    // Приоритет 2: Датчики движения (ТЗ 2.0)
    // Защита от дребезга и удержание сигнала движения с помощью TOF
    L_Motion_Timers[L_i](IN := VI_Motion_Sensors[L_i], PT := T#5m, VI_System_Time_MS := VI_System_Time_MS);
    
    // Сброс ручного переопределения, когда комната становится пустой (задний фронт таймера движения)
    IF L_Prev_Motion_Q[L_i] AND NOT L_Motion_Timers[L_i].Q THEN
        L_Manual_Override[L_i] := FALSE;
    END_IF;
    L_Prev_Motion_Q[L_i] := L_Motion_Timers[L_i].Q;

    IF L_Motion_Timers[L_i].Q THEN
        IF NOT L_Manual_Override[L_i] THEN
            L_Light_States[L_i] := TRUE;
        END_IF;
    ELSE
        // Выключаем свет только если нет ручного переопределения
        IF NOT L_Manual_Override[L_i] THEN
            L_Light_States[L_i] := FALSE;
        END_IF;
    END_IF;

    // Приоритет 3: Симуляция (только в режиме Away)
    IF L_Effective_Scenario = E_SCENARIO_TYPE.SCENARIO_AWAY AND L_Effective_Simulation_Active THEN
        L_Light_States[L_i] := VI_Simulation_Lights[L_i];
    END_IF;

    // Приоритет 4: Ручное управление и правила
    IF VI_Manual_Light_Override[L_i] > 0 THEN
        VO_Lighting_Levels[L_i] := VI_Manual_Light_Override[L_i];
    ELSIF L_Rule_Light_Active THEN
        VO_Lighting_Levels[L_i] := L_Rule_Light_Val;
    ELSE
        VO_Lighting_Levels[L_i] := SEL(L_Light_States[L_i], 0, L_Base_Light);
    END_IF;
    
    // 5. Мокрые зоны
    IF VI_Wet_Zone_Map[L_i] AND L_Wet_Zone_Idx <= GVL_CONSTANTS.C_MAX_WET_ZONES THEN
        VO_Wet_Zone_Light_Active[L_Wet_Zone_Idx] := (VO_Lighting_Levels[L_i] > 10);
        L_Wet_Zone_Idx := L_Wet_Zone_Idx + 1;
    END_IF;
END_FOR;

// 3. Управление шторами
FOR L_i := 1 TO GVL_CONSTANTS.C_MAX_BLINDS DO
    L_Rule_Blinds_Active := FALSE;
    L_Rule_Blinds_Val := 0;
    
    // Проверка правил
    FOR L_j := 1 TO GVL_CONSTANTS.C_MAX_RULES DO
        IF VI_Rule_Actions[L_j].Active AND VI_Rule_Actions[L_j].Target_ID = L_i THEN
            IF VI_Rule_Actions[L_j].Action_Type = E_Rule_Action_Type.ACTION_SET_BLINDS THEN
                L_Rule_Blinds_Active := TRUE;
                L_Rule_Blinds_Val := REAL_TO_BYTE(VI_Rule_Actions[L_j].Value);
            END_IF;
        END_IF;
    END_FOR;

    // Приоритет 1: Ручное управление
    IF VI_Manual_Blinds_Override[L_i] > 0 THEN
        VO_Blinds_Positions[L_i] := VI_Manual_Blinds_Override[L_i];
    // Приоритет 2: Правила
    ELSIF L_Rule_Blinds_Active THEN
        VO_Blinds_Positions[L_i] := L_Rule_Blinds_Val;
    // Приоритет 3: Сценарий
    ELSE
        VO_Blinds_Positions[L_i] := L_Base_Blinds;
    END_IF;
END_FOR;

// >>> BULK_SYNC_ANCHOR: FB_Lighting_Blinds_Manager <<<
          
END_FUNCTION_BLOCK

FUNCTION_BLOCK FB_Trace_Logger
  VAR_INPUT
    VI_Event_Code : INT;
    VI_System_Time : UDINT;
  END_VAR

            GVL_TRACE.G_Trace_Index := GVL_TRACE.G_Trace_Index + 1;
IF GVL_TRACE.G_Trace_Index > GVL_TRACE.G_Trace_Max THEN
    GVL_TRACE.G_Trace_Index := 1;
END_IF;

GVL_TRACE.G_Trace_Time[GVL_TRACE.G_Trace_Index] := VI_System_Time;
GVL_TRACE.G_Trace_Code[GVL_TRACE.G_Trace_Index] := VI_Event_Code;
          
END_FUNCTION_BLOCK

FUNCTION_BLOCK FB_Heating_System_Manager
  VAR_INPUT
    VI_Preheat_Request : BOOL;
    L_Climate_Zone_ID : INT;
    VI_System_Mode : E_System_Operating_Mode;
    VI_System_Time_MS : UDINT;
    VI_Current_TOD : TOD;
    VI_IsActivePLC : BOOL;
    VI_Outdoor_Temp : REAL;
    VI_Config : ST_Heating_Config;
    VI_Tariff : ST_Tariff_Config;
    VI_Current_Hour : UINT;
    VI_Boiler_Stop : BOOL;
    VI_DHW_Heating_Demand : BOOL;
    VI_DHW_Target_Temp : REAL;
    VI_Current_Scenario : E_SCENARIO_TYPE;
    VI_Emergency_Stop : BOOL;
    VI_Gas_Safety_Stop : BOOL;
    VI_Boiler_Error_Status : ARRAY[1..GVL_CONSTANTS.C_MAX_BOILERS] OF BOOL;
    VI_Boiler_OT_Online : ARRAY[1..GVL_CONSTANTS.C_MAX_BOILERS] OF BOOL;
    VI_Boiler_Modulation : ARRAY[1..GVL_CONSTANTS.C_MAX_BOILERS] OF REAL;
  END_VAR
  VAR_OUTPUT
    VO_Manifold_Valves : ARRAY[1..GVL_CONSTANTS.C_MAX_MANIFOLDS] OF REAL;
    VO_Manifold_Pumps : ARRAY[1..GVL_CONSTANTS.C_MAX_MANIFOLDS] OF BOOL;
    VO_Zone_Valves : ARRAY[1..GVL_CONSTANTS.C_MAX_HEATING_CIRCUITS] OF BOOL;
    VO_Boiler_OT_Enable : ARRAY[1..GVL_CONSTANTS.C_MAX_BOILERS] OF BOOL;
    VO_Boiler_OT_Setpoint : ARRAY[1..GVL_CONSTANTS.C_MAX_BOILERS] OF REAL;
    VO_Backup_Circulation_Pump : BOOL;
    VO_Electric_Heater_Enable : BOOL;
    VO_Freeze_Risk_Status : BOOL;
    VO_Status : ARRAY[1..GVL_CONSTANTS.C_MAX_MANIFOLDS] OF ST_Manifold_Status;
    VO_Boiler_Status : ARRAY[1..GVL_CONSTANTS.C_MAX_BOILERS] OF ST_Boiler_Status;
  END_VAR
  VAR_IN_OUT
    VI_Floor_Temps : ARRAY[1..GVL_CONSTANTS.C_MAX_HEATING_CIRCUITS] OF REAL;
    VI_Room_Temps : ARRAY[1..16] OF REAL;
    VI_Manifold_Pressures : ARRAY[1..GVL_CONSTANTS.C_MAX_MANIFOLDS] OF REAL;
    VI_Manifold_Currents : ARRAY[1..GVL_CONSTANTS.C_MAX_MANIFOLDS] OF REAL;
    VI_Manifold_Temps_Supply : ARRAY[1..GVL_CONSTANTS.C_MAX_MANIFOLDS] OF REAL;
    VI_Manifold_Temps_Return : ARRAY[1..GVL_CONSTANTS.C_MAX_MANIFOLDS] OF REAL;
    VI_Boiler_Flame_Status : ARRAY[1..GVL_CONSTANTS.C_MAX_BOILERS] OF BOOL;
    VI_Zone_Configs : ARRAY[1..GVL_CONSTANTS.C_MAX_HEATING_CIRCUITS] OF ST_FloorHeating_Circuit_Config;
    VI_Rule_Actions : ARRAY[1..GVL_CONSTANTS.C_MAX_RULES] OF ST_Rule_Action;
    VI_IO_Modules_Online : ARRAY[1..GVL_CONSTANTS.C_MAX_MODULES] OF BOOL;
    VI_Scenario_Configs : ARRAY[1..GVL_CONSTANTS.C_MAX_SCENARIOS] OF ST_Scenario_Config;
    VI_Manifold_End_Switches : ARRAY[1..GVL_CONSTANTS.C_MAX_MANIFOLDS] OF BOOL;
    VI_Valve_Test_Config : ARRAY[1..GVL_CONSTANTS.C_MAX_MANIFOLDS] OF ST_Valve_Test_Config;
  END_VAR
  VAR
    L_Lead_Boiler : BYTE := 1;
    L_i : INT;
    L_j : INT;
    L_Target_Supply_Temp : REAL;
    L_Demand_Power : REAL;
    L_Any_Zone_Active : ARRAY[1..GVL_CONSTANTS.C_MAX_MANIFOLDS] OF BOOL;
    L_Prev_Scenario : E_SCENARIO_TYPE;
    L_Scenario_Adjust : REAL;
    L_Target_Scenario_Adjust : REAL;
    L_Transition_Temp : FB_Scenario_Transition_Controller;
    fbValveTestManager : FB_Valve_Test_Manager;
    L_IO_Failsafe_Active : BOOL;
    L_Freeze_Mode_Active : BOOL;
    L_Freeze_Target_Supply : REAL;
    L_Min_Supply_Temp : REAL;
    L_Policy_Degraded : BOOL;
    L_Any_Sensor_Error : BOOL;
    L_Any_Subsystem_Degraded : BOOL;
    L_Adaptive_Max_Delta : REAL;
    L_Adaptive_Effective_Delta : REAL;
    L_Adaptive_Correction : REAL;
    fbAdaptiveTarget : FB_Heating_Adaptive_Target;
    fbSafetyGate : FB_Heating_Safety_Gate;
    fbCircuitControl : FB_Heating_Circuit_Control;
    fbManifoldControl : FB_Heating_Manifold_Control;
    fbBoilerControl : FB_Heating_Boiler_Control;
  END_VAR

            // ==============================================================================
// Блок управления системой отопления (Heating System Manager)
// Назначение:
// - Публичный фасад системы отопления.
// - Оркестрация доменных FB отопления.
// - Проекция безопасных состояний на физические выходы.
// - Интеграция с Rule Engine, HMI status и GVL_STATE.
// ==============================================================================



// ========================================
// Policy and fault pre-scan
// ========================================
L_Policy_Degraded := (VI_System_Mode = E_System_Operating_Mode.MODE_DEGRADED);

GVL_STATE.G_Heating_IO_Fault := FALSE;
GVL_STATE.G_Heating_Sensor_Fault := FALSE;
GVL_STATE.G_Heating_Subsystem_Degraded := FALSE;
L_Any_Sensor_Error := FALSE;
L_Any_Subsystem_Degraded := FALSE;

L_IO_Failsafe_Active := FALSE;
FOR L_i := 1 TO GVL_CONSTANTS.C_MAX_MODULES DO
    IF NOT VI_IO_Modules_Online[L_i] THEN
        L_IO_Failsafe_Active := TRUE;
        GVL_STATE.G_Heating_IO_Fault := TRUE;
        GVL_STATE.G_Heating_Subsystem_Degraded := TRUE;
        EXIT;
    END_IF;
END_FOR;

fbSafetyGate(
    VI_System_Mode := VI_System_Mode,
    VI_Emergency_Stop := VI_Emergency_Stop,
    VI_Gas_Safety_Stop := VI_Gas_Safety_Stop,
    VI_IO_Failsafe_Active := L_IO_Failsafe_Active,
    VI_Outdoor_Temp := VI_Outdoor_Temp,
    VI_Freeze_Threshold := VI_Config.Freeze_Threshold,
    VI_Floor_Temps := VI_Floor_Temps,
    VO_Freeze_Mode_Active => L_Freeze_Mode_Active,
    VO_Freeze_Target_Supply => L_Freeze_Target_Supply
);

// ========================================
// Safe-state output projection
// ========================================
VO_Backup_Circulation_Pump := FALSE;
VO_Electric_Heater_Enable := FALSE;
VO_Freeze_Risk_Status := FALSE;

IF fbSafetyGate.VO_Block_Normal_Heating THEN
    FOR L_i := 1 TO GVL_CONSTANTS.C_MAX_HEATING_CIRCUITS DO
        VO_Zone_Valves[L_i] := FALSE;
    END_FOR;

    FOR L_i := 1 TO GVL_CONSTANTS.C_MAX_MANIFOLDS DO
        IF fbSafetyGate.VO_IO_Failsafe_Active AND L_Freeze_Mode_Active THEN
            VO_Manifold_Pumps[L_i] := TRUE;
            VO_Manifold_Valves[L_i] := 35.0;
        ELSE
            VO_Manifold_Pumps[L_i] := FALSE;
            VO_Manifold_Valves[L_i] := 0.0;
        END_IF;
    END_FOR;

    FOR L_i := 1 TO GVL_CONSTANTS.C_MAX_BOILERS DO
        VO_Boiler_OT_Enable[L_i] := FALSE;
        VO_Boiler_OT_Setpoint[L_i] := 0.0;
        VO_Boiler_Status[L_i].Warning := FALSE;
        VO_Boiler_Status[L_i].Error := TRUE;
    END_FOR;

    IF fbSafetyGate.VO_Gas_Safety_Active AND L_Freeze_Mode_Active THEN
        VO_Backup_Circulation_Pump := TRUE;
        L_Min_Supply_Temp := 1000.0;
        FOR L_i := 1 TO GVL_CONSTANTS.C_MAX_MANIFOLDS DO
            IF VI_Manifold_Temps_Supply[L_i] < L_Min_Supply_Temp THEN
                L_Min_Supply_Temp := VI_Manifold_Temps_Supply[L_i];
            END_IF;
        END_FOR;
        IF L_Min_Supply_Temp > 900.0 THEN
            L_Min_Supply_Temp := 0.0;
        END_IF;

        IF L_Min_Supply_Temp < (L_Freeze_Target_Supply - 1.0) THEN
            VO_Electric_Heater_Enable := TRUE;
        ELSIF L_Min_Supply_Temp > (L_Freeze_Target_Supply + 1.0) THEN
            VO_Electric_Heater_Enable := FALSE;
        END_IF;

        // При защёлкнутой газовой аварии оператор должен видеть, что система живёт в деградированном anti-freeze режиме.
        VO_Freeze_Risk_Status := TRUE;
    END_IF;

    IF fbSafetyGate.VO_IO_Failsafe_Active AND L_Freeze_Mode_Active THEN
        IF VI_Boiler_OT_Online[1] AND NOT VI_Boiler_Error_Status[1] THEN
            VO_Boiler_OT_Enable[1] := TRUE;
            VO_Boiler_OT_Setpoint[1] := L_Freeze_Target_Supply;
        END_IF;
    END_IF;

    RETURN;
END_IF;

// --- ADAPTIVE TARGET ---
fbAdaptiveTarget(
    VI_Base_Target_Supply_Temp := L_Target_Supply_Temp,
    VI_Global_Target_Temperature := GVL_STATE.G_Target_Temperature,
    VI_Zone_Configs := VI_Zone_Configs,
    VI_Floor_Temps := VI_Floor_Temps,
    VI_Room_Temps := VI_Room_Temps,
    VO_Target_Supply_Temp => L_Target_Supply_Temp,
    VO_Adaptive_Correction => L_Adaptive_Correction,
    VO_Adaptive_Effective_Delta => L_Adaptive_Effective_Delta,
    VO_Adaptive_Max_Delta => L_Adaptive_Max_Delta
);

// --- CIRCUIT CONTROL ---
fbCircuitControl(
    VI_System_Time_MS := VI_System_Time_MS,
    VI_Current_Hour := VI_Current_Hour,
    VI_IsActivePLC := VI_IsActivePLC,
    VI_Config := VI_Config,
    VI_Tariff := VI_Tariff,
    VI_Scenario_Adjust := L_Scenario_Adjust,
    VI_Zone_Configs := VI_Zone_Configs,
    VI_Floor_Temps := VI_Floor_Temps,
    VI_Room_Temps := VI_Room_Temps,
    VI_Rule_Actions := VI_Rule_Actions,
    VO_Zone_Valves => VO_Zone_Valves,
    VO_Heating_Sensor_Fault => L_Any_Sensor_Error
);

GVL_STATE.G_Heating_Sensor_Fault := L_Any_Sensor_Error;

// --- MANIFOLD DEMAND MAP ---
FOR L_i := 1 TO GVL_CONSTANTS.C_MAX_MANIFOLDS DO
    L_Any_Zone_Active[L_i] := FALSE;
END_FOR;

FOR L_i := 1 TO GVL_CONSTANTS.C_MAX_HEATING_CIRCUITS DO
    IF VO_Zone_Valves[L_i] THEN
        L_j := VI_Zone_Configs[L_i].manifold_id;
        IF L_j >= 1 AND L_j <= GVL_CONSTANTS.C_MAX_MANIFOLDS THEN
            L_Any_Zone_Active[L_j] := TRUE;
        END_IF;
    END_IF;
END_FOR;

// --- MANIFOLD CONTROL ---
fbManifoldControl(
    VI_System_Time_MS := VI_System_Time_MS,
    VI_IsActivePLC := VI_IsActivePLC,
    VI_DHW_Heating_Demand := VI_DHW_Heating_Demand,
    VI_Freeze_Mode_Active := L_Freeze_Mode_Active,
    VI_Target_Supply_Temp := L_Target_Supply_Temp,
    VI_Any_Zone_Active := L_Any_Zone_Active,
    VI_Manifold_Pressures := VI_Manifold_Pressures,
    VI_Manifold_Currents := VI_Manifold_Currents,
    VI_Manifold_Temps_Supply := VI_Manifold_Temps_Supply,
    VI_Manifold_Temps_Return := VI_Manifold_Temps_Return,
    VO_Manifold_Pumps => VO_Manifold_Pumps,
    VO_Manifold_Valves => VO_Manifold_Valves,
    VO_Status => VO_Status
);

// --- VALVE TEST OVERRIDE ---
fbValveTestManager(
    VI_System_Time_MS := VI_System_Time_MS,
    VI_IsActivePLC := VI_IsActivePLC,
    VI_Valve_Currents := VI_Manifold_Currents,
    VI_Valve_End_Switches := VI_Manifold_End_Switches,
    VI_Config := VI_Valve_Test_Config
);

IF fbValveTestManager.VO_Test_Active THEN
    L_i := fbValveTestManager.VO_Current_Valve;
    IF L_i >= 1 AND L_i <= GVL_CONSTANTS.C_MAX_MANIFOLDS THEN
        IF fbValveTestManager.VO_Valve_Cmd[L_i] THEN
            VO_Manifold_Valves[L_i] := 100.0;
        ELSE
            VO_Manifold_Valves[L_i] := 0.0;
        END_IF;
        VO_Manifold_Pumps[L_i] := FALSE; // Отключаем насос при тестировании клапана
    END_IF;
END_IF;

// --- BOILER CONTROL ---
fbBoilerControl(
    VI_System_Time_MS := VI_System_Time_MS,
    VI_IsActivePLC := VI_IsActivePLC,
    VI_DHW_Heating_Demand := VI_DHW_Heating_Demand,
    VI_DHW_Target_Temp := VI_DHW_Target_Temp,
    VI_Target_Supply_Temp := L_Target_Supply_Temp,
    VI_Freeze_Mode_Active := L_Freeze_Mode_Active,
    VI_Policy_Degraded := L_Policy_Degraded,
    VI_Manifold_Pumps := VO_Manifold_Pumps,
    VI_Manifold_Valves := VO_Manifold_Valves,
    VI_Boiler_Flame_Status := VI_Boiler_Flame_Status,
    VI_Boiler_Error_Status := VI_Boiler_Error_Status,
    VI_Boiler_OT_Online := VI_Boiler_OT_Online,
    VI_Boiler_Modulation := VI_Boiler_Modulation,
    VO_Boiler_OT_Enable => VO_Boiler_OT_Enable,
    VO_Boiler_OT_Setpoint => VO_Boiler_OT_Setpoint,
    VO_Boiler_Status => VO_Boiler_Status,
    VO_Any_Subsystem_Degraded => L_Any_Subsystem_Degraded,
    VO_Lead_Boiler => L_Lead_Boiler,
    VO_Demand_Power => L_Demand_Power
);

GVL_STATE.G_Heating_Subsystem_Degraded := L_Any_Subsystem_Degraded;

// >>> BULK_SYNC_ANCHOR: FB_Heating_System_Manager <<<
          
END_FUNCTION_BLOCK

FUNCTION_BLOCK FB_Water_Leakage_Manager
  VAR_INPUT
    VI_System_Time_MS : UDINT;
    VI_IsActivePLC : BOOL;
    VI_Config : ST_Flood_Global_Config;
  END_VAR
  VAR_OUTPUT
    VO_Status_Msg : STRING(200);
    VO_Leak_Detected : BOOL;
    VO_Leak_Warning_Level : BOOL;
  END_VAR
  VAR_IN_OUT
    VI_Sensors : ARRAY[1..GVL_CONSTANTS.C_MAX_FLOOD_SENSORS] OF BOOL;
  END_VAR
  VAR
    L_i : INT;
    L_Sensor_Timers : ARRAY[1..GVL_CONSTANTS.C_MAX_FLOOD_SENSORS] OF FB_System_Timer;
    L_Any_Leak : BOOL;
    L_Any_Warning : BOOL;
  END_VAR

            IF NOT VI_IsActivePLC THEN RETURN; END_IF;

L_Any_Leak := FALSE;
L_Any_Warning := FALSE;

FOR L_i := 1 TO GVL_CONSTANTS.C_MAX_FLOOD_SENSORS DO
    L_Sensor_Timers[L_i](
        IN := VI_Sensors[L_i],
        PT := TO_TIME(VI_Config.min_duration_ms + VI_Config.warning_duration_ms),
        VI_System_Time_MS := VI_System_Time_MS
    );

    IF L_Sensor_Timers[L_i].ET >= TO_TIME(VI_Config.min_duration_ms) THEN
        L_Any_Warning := TRUE;

        IF L_Sensor_Timers[L_i].Q THEN
            L_Any_Leak := TRUE;
        END_IF;
    END_IF;
END_FOR;

// Health signals
VO_Leak_Detected := L_Any_Leak;
VO_Leak_Warning_Level := L_Any_Warning;

// Status
IF L_Any_Leak THEN
    VO_Status_Msg := 'АВАРИЯ: ПРОТЕЧКА ВОДЫ.';
ELSIF L_Any_Warning THEN
    VO_Status_Msg := 'ПРЕДУПРЕЖДЕНИЕ: ОБНАРУЖЕНА ВОДА.';
ELSE
    VO_Status_Msg := 'Система контроля протечек в норме';
END_IF;
// >>> BULK_SYNC_ANCHOR: FB_Water_Leakage_Manager <<<
          
END_FUNCTION_BLOCK

FUNCTION_BLOCK FB_Heating_Policy_Observer
  VAR_INPUT
    VI_Zone_Occupied : ARRAY[1..GVL_CONSTANTS.C_MAX_ZONES] OF BOOL;
    VI_Zone_Last_Motion_TS : ARRAY[1..GVL_CONSTANTS.C_MAX_ZONES] OF UDINT;
    VI_System_Time_MS : UDINT;
    VI_Zone_Permanent_Use : ARRAY[1..GVL_CONSTANTS.C_MAX_ZONES] OF BOOL;
    VI_Zone_Guest_Preheat : ARRAY[1..GVL_CONSTANTS.C_MAX_ZONES] OF BOOL;
    VI_Behavior_Mode : E_Behavior_Mode;
  END_VAR
  VAR_OUTPUT
    VO_Zone_Empty_Duration_MS : ARRAY[1..GVL_CONSTANTS.C_MAX_ZONES] OF UDINT;
    VO_Zone_Policy_Class : ARRAY[1..GVL_CONSTANTS.C_MAX_ZONES] OF INT;
    VO_Zone_Target_Adjustment : ARRAY[1..GVL_CONSTANTS.C_MAX_ZONES] OF REAL;
    VO_Zone_Priority_Bias : ARRAY[1..GVL_CONSTANTS.C_MAX_ZONES] OF REAL;
  END_VAR
  VAR
    L_i : INT;
    L_Long_Threshold : UDINT := 86400000;
    L_Away_Mode : BOOL;
  END_VAR

            L_Away_Mode := (VI_Behavior_Mode = BEHAVIOR_AWAY);

FOR L_i := 1 TO GVL_CONSTANTS.C_MAX_ZONES DO

    // compute empty duration
    IF VI_Zone_Occupied[L_i] THEN
        VO_Zone_Empty_Duration_MS[L_i] := 0;
    ELSE
        VO_Zone_Empty_Duration_MS[L_i] := VI_System_Time_MS - VI_Zone_Last_Motion_TS[L_i];
    END_IF;

    // policy classification
    // Guest/preheat has priority even in AWAY mode.
    IF VI_Zone_Guest_Preheat[L_i] THEN
        VO_Zone_Policy_Class[L_i] := 3; // guest

    ELSIF VI_Zone_Occupied[L_i] THEN
        VO_Zone_Policy_Class[L_i] := 0; // comfort

    ELSIF VI_Zone_Permanent_Use[L_i] AND (NOT L_Away_Mode) THEN
        VO_Zone_Policy_Class[L_i] := 4; // permanent mild eco

    ELSIF VO_Zone_Empty_Duration_MS[L_i] >= L_Long_Threshold THEN
        VO_Zone_Policy_Class[L_i] := 2; // deep eco

    ELSE
        VO_Zone_Policy_Class[L_i] := 1; // mild eco
    END_IF;

    // observe-only target adjustment (no effect yet)
    CASE VO_Zone_Policy_Class[L_i] OF
        0: // comfort
            VO_Zone_Target_Adjustment[L_i] := 0.0;
            VO_Zone_Priority_Bias[L_i] := 1.0;

        1: // mild eco
            VO_Zone_Target_Adjustment[L_i] := -1.0;
            VO_Zone_Priority_Bias[L_i] := 0.8;

        2: // deep eco
            VO_Zone_Target_Adjustment[L_i] := -3.0;
            VO_Zone_Priority_Bias[L_i] := 0.5;

        3: // guest preheat
            VO_Zone_Target_Adjustment[L_i] := 0.0;
            VO_Zone_Priority_Bias[L_i] := 1.5;

        4: // permanent-use mild eco
            VO_Zone_Target_Adjustment[L_i] := -0.5;
            VO_Zone_Priority_Bias[L_i] := 0.9;

    END_CASE;

END_FOR;
          
END_FUNCTION_BLOCK

FUNCTION_BLOCK FB_Simulation_Manager
  VAR_INPUT
    VI_System_Time_MS : UDINT;
    VI_IsActivePLC : BOOL;
    VI_Scenario : E_SCENARIO_TYPE;
    VI_Config : ST_Scenario_Config;
  END_VAR
  VAR_OUTPUT
    VO_Sim_Lights : ARRAY[1..32] OF BOOL;
    VO_Sim_Active : BOOL;
    VO_Sim_Water_Leak : ARRAY[1..GVL_CONSTANTS.C_MAX_FLOOD_SENSORS] OF BOOL;
    VO_Sim_Gas_Leak : ARRAY[1..GVL_CONSTANTS.C_MAX_METHANE_SENSORS] OF REAL;
  END_VAR
  VAR
    L_Random : FB_Random_Generator;
    L_Last_Toggle : UDINT;
    L_i : INT;
    L_Rand_Val : UDINT;
    L_Test_Mode : BOOL := FALSE;
  END_VAR

            IF VI_Scenario = E_SCENARIO_TYPE.SCENARIO_AWAY AND VI_Config.Presence_Simulation_Enabled THEN
    VO_Sim_Active := TRUE;
    
    // Переключаем свет каждые 30 минут
    IF (VI_System_Time_MS - L_Last_Toggle) >= (GVL_CONSTANTS.C_MS_IN_MINUTE * 30) THEN
        L_Last_Toggle := VI_System_Time_MS;
        
        FOR L_i := 1 TO 32 DO
            L_Rand_Val := 1;
            VO_Sim_Lights[L_i] := (L_Rand_Val > 80); // 20% шанс включения
        END_FOR;
    END_IF;
ELSE
    VO_Sim_Active := FALSE;
    FOR L_i := 1 TO 32 DO VO_Sim_Lights[L_i] := FALSE; END_FOR;
END_IF;

// Симуляция аварий в тестовом режиме
IF L_Test_Mode THEN
    // Генерация случайных протечек (очень редко)
    L_Rand_Val := 1;
    IF L_Rand_Val = 42 THEN
        VO_Sim_Water_Leak[1] := TRUE;
    END_IF;
    
    // Симуляция утечки газа
    L_Rand_Val := 1;
    IF L_Rand_Val = 77 THEN
        VO_Sim_Gas_Leak[1] := 15.0; // 15% LEL
    END_IF;
ELSE
    FOR L_i := 1 TO GVL_CONSTANTS.C_MAX_FLOOD_SENSORS DO VO_Sim_Water_Leak[L_i] := FALSE; END_FOR;
    FOR L_i := 1 TO GVL_CONSTANTS.C_MAX_METHANE_SENSORS DO VO_Sim_Gas_Leak[L_i] := 0.0; END_FOR;
END_IF;
// >>> BULK_SYNC_ANCHOR: FB_Simulation_Manager <<<
          
END_FUNCTION_BLOCK

FUNCTION_BLOCK FB_Boiler_OpenTherm_Interface
  VAR_INPUT
    VI_Enable : ARRAY[1..GVL_CONSTANTS.C_MAX_BOILERS] OF BOOL;
    VI_Setpoint : ARRAY[1..GVL_CONSTANTS.C_MAX_BOILERS] OF REAL;
    VI_OT_Online : ARRAY[1..GVL_CONSTANTS.C_MAX_BOILERS] OF BOOL;
    VI_OT_Error : ARRAY[1..GVL_CONSTANTS.C_MAX_BOILERS] OF BOOL;
  END_VAR
  VAR_OUTPUT
    VO_OT_Enable : ARRAY[1..GVL_CONSTANTS.C_MAX_BOILERS] OF BOOL;
    VO_OT_Setpoint : ARRAY[1..GVL_CONSTANTS.C_MAX_BOILERS] OF REAL;
    VO_OT_Command_Valid : ARRAY[1..GVL_CONSTANTS.C_MAX_BOILERS] OF BOOL;
  END_VAR
  VAR
    L_i : INT;
  END_VAR

            FOR L_i := 1 TO GVL_CONSTANTS.C_MAX_BOILERS DO
    VO_OT_Enable[L_i] := FALSE;
    VO_OT_Setpoint[L_i] := 0.0;
    VO_OT_Command_Valid[L_i] := FALSE;

    IF VI_Enable[L_i] AND VI_OT_Online[L_i] AND NOT VI_OT_Error[L_i] THEN
        VO_OT_Enable[L_i] := TRUE;
        VO_OT_Setpoint[L_i] := LIMIT(20.0, VI_Setpoint[L_i], 80.0);
        VO_OT_Command_Valid[L_i] := TRUE;
    END_IF;
END_FOR;
          
END_FUNCTION_BLOCK

FUNCTION_BLOCK FB_Heating_Adaptive_Target
  VAR_INPUT
    VI_Base_Target_Supply_Temp : REAL;
    VI_Global_Target_Temperature : REAL;
  END_VAR
  VAR_OUTPUT
    VO_Target_Supply_Temp : REAL;
    VO_Adaptive_Correction : REAL;
    VO_Adaptive_Effective_Delta : REAL;
    VO_Adaptive_Max_Delta : REAL;
  END_VAR
  VAR_IN_OUT
    VI_Zone_Configs : ARRAY[1..GVL_CONSTANTS.C_MAX_HEATING_CIRCUITS] OF ST_FloorHeating_Circuit_Config;
    VI_Floor_Temps : ARRAY[1..GVL_CONSTANTS.C_MAX_HEATING_CIRCUITS] OF REAL;
    VI_Room_Temps : ARRAY[1..16] OF REAL;
  END_VAR
  VAR
    L_Adaptive_Zone_i : INT;
    L_Adaptive_Delta : REAL;
    L_Adaptive_Weighted_Sum : REAL;
    L_Adaptive_Weight_Total : REAL;
    L_Adaptive_Weight : REAL;
  END_VAR

            // ==============================================================================
// Adaptive target calculation for heating supply temperature
//
// Internal refactoring helper for FB_Heating_System_Manager.
// The manager remains the public facade; this block only extracts the adaptive
// target calculation section to reduce large-file edit risk.
// ==============================================================================



VO_Target_Supply_Temp := VI_Base_Target_Supply_Temp;
VO_Adaptive_Max_Delta := 0.0;
L_Adaptive_Weighted_Sum := 0.0;
L_Adaptive_Weight_Total := 0.0;
VO_Adaptive_Effective_Delta := 0.0;
VO_Adaptive_Correction := 0.0;

// Global arbitration target is applied before adaptive correction.
IF VI_Global_Target_Temperature > 0.0 THEN
    VO_Target_Supply_Temp := VI_Global_Target_Temperature;
END_IF;

// Final adaptive refinement layer.
FOR L_Adaptive_Zone_i := 1 TO GVL_CONSTANTS.C_MAX_HEATING_CIRCUITS DO
    IF VI_Zone_Configs[L_Adaptive_Zone_i].zone >= 1 AND VI_Zone_Configs[L_Adaptive_Zone_i].zone <= 8 THEN
        CASE VI_Zone_Configs[L_Adaptive_Zone_i].control_type OF
            0:
                L_Adaptive_Delta :=
                    VI_Zone_Configs[L_Adaptive_Zone_i].design_temp -
                    VI_Floor_Temps[L_Adaptive_Zone_i];
                L_Adaptive_Weight := 0.6;
            1, 2:
                L_Adaptive_Delta :=
                    VI_Zone_Configs[L_Adaptive_Zone_i].design_temp -
                    VI_Room_Temps[VI_Zone_Configs[L_Adaptive_Zone_i].zone];
                L_Adaptive_Weight := 1.0;
            ELSE
                L_Adaptive_Delta :=
                    VI_Zone_Configs[L_Adaptive_Zone_i].design_temp -
                    VI_Room_Temps[VI_Zone_Configs[L_Adaptive_Zone_i].zone];
                L_Adaptive_Weight := 0.8;
        END_CASE;

        IF VI_Zone_Configs[L_Adaptive_Zone_i].zone >= 1 AND VI_Zone_Configs[L_Adaptive_Zone_i].zone <= 4 THEN
            L_Adaptive_Weight := L_Adaptive_Weight * 1.2;
        ELSIF VI_Zone_Configs[L_Adaptive_Zone_i].zone >= 9 THEN
            L_Adaptive_Weight := L_Adaptive_Weight * 0.7;
        END_IF;

        IF L_Adaptive_Weight > 2.0 THEN
            L_Adaptive_Weight := 2.0;
        ELSIF L_Adaptive_Weight < 0.2 THEN
            L_Adaptive_Weight := 0.2;
        END_IF;

        IF L_Adaptive_Delta > VO_Adaptive_Max_Delta THEN
            VO_Adaptive_Max_Delta := L_Adaptive_Delta;
        END_IF;

        L_Adaptive_Weighted_Sum := L_Adaptive_Weighted_Sum + (L_Adaptive_Delta * L_Adaptive_Weight);
        L_Adaptive_Weight_Total := L_Adaptive_Weight_Total + L_Adaptive_Weight;
    END_IF;
END_FOR;

IF L_Adaptive_Weight_Total > 0.0 THEN
    VO_Adaptive_Effective_Delta := L_Adaptive_Weighted_Sum / L_Adaptive_Weight_Total;
END_IF;

IF VO_Adaptive_Effective_Delta > 1.5 THEN
    VO_Adaptive_Correction := 2.0;
ELSIF VO_Adaptive_Effective_Delta > 0.7 THEN
    VO_Adaptive_Correction := 1.0;
ELSIF VO_Adaptive_Effective_Delta < -1.5 THEN
    VO_Adaptive_Correction := -2.0;
ELSIF VO_Adaptive_Effective_Delta < -0.7 THEN
    VO_Adaptive_Correction := -1.0;
ELSE
    VO_Adaptive_Correction := 0.0;
END_IF;

IF VO_Adaptive_Max_Delta > 2.5 AND VO_Adaptive_Correction < 2.0 THEN
    VO_Adaptive_Correction := 2.0;
END_IF;

VO_Target_Supply_Temp := VO_Target_Supply_Temp + VO_Adaptive_Correction;

IF VO_Target_Supply_Temp < 20.0 THEN
    VO_Target_Supply_Temp := 20.0;
ELSIF VO_Target_Supply_Temp > 45.0 THEN
    VO_Target_Supply_Temp := 45.0;
END_IF;

// >>> BULK_SYNC_ANCHOR: FB_Heating_Adaptive_Target <<<
          
END_FUNCTION_BLOCK

FUNCTION_BLOCK FB_Ownership_Watchdog
  VAR_INPUT
    VI_Gas_Level : REAL;
    VI_Gas_Alarm : BOOL;
    VI_Leak_Alarm : BOOL;
    VI_Smoke_Alarm : BOOL;
  END_VAR
  VAR_OUTPUT
    VO_Ownership_Violation : BOOL;
  END_VAR
  VAR
    L_Last_Gas_Alarm : BOOL;
    L_Last_Leak_Alarm : BOOL;
    L_Last_Smoke_Alarm : BOOL;
  END_VAR

            VO_Ownership_Violation := FALSE;

// Gas: signal present, alarm disappeared
IF (VI_Gas_Level > 20.0) AND L_Last_Gas_Alarm AND (NOT VI_Gas_Alarm) THEN
    VO_Ownership_Violation := TRUE;
END_IF;

// Leak: once latched should not drop instantly
IF L_Last_Leak_Alarm AND (NOT VI_Leak_Alarm) THEN
    VO_Ownership_Violation := TRUE;
END_IF;

// Smoke: same rule
IF L_Last_Smoke_Alarm AND (NOT VI_Smoke_Alarm) THEN
    VO_Ownership_Violation := TRUE;
END_IF;

L_Last_Gas_Alarm := VI_Gas_Alarm;
L_Last_Leak_Alarm := VI_Leak_Alarm;
L_Last_Smoke_Alarm := VI_Smoke_Alarm;
          
END_FUNCTION_BLOCK

FUNCTION_BLOCK FB_Safety_Workflow_Manager
  VAR_INPUT
    VI_System_Time_MS : UDINT;
    VI_Water_Selective_Recover : BOOL;
    VI_Gas_Selective_Recover : BOOL;
    VI_Water_Valve_Test_Open : BOOL;
    VI_Water_Valve_Test_Close : BOOL;
    VI_Water_Valve_Test_Confirm : BOOL;
    VI_Gas_Valve_Test_Open : BOOL;
    VI_Gas_Valve_Test_Close : BOOL;
    VI_Gas_Valve_Test_Confirm : BOOL;
  END_VAR
  VAR_OUTPUT
    VO_Water_Selective_Recover_Edge : BOOL;
    VO_Gas_Selective_Recover_Edge : BOOL;
    VO_Water_Valve_Test_Open_Edge : BOOL;
    VO_Water_Valve_Test_Close_Edge : BOOL;
    VO_Water_Valve_Test_Confirm_Edge : BOOL;
    VO_Gas_Valve_Test_Open_Edge : BOOL;
    VO_Gas_Valve_Test_Close_Edge : BOOL;
    VO_Gas_Valve_Test_Confirm_Edge : BOOL;
    VO_Water_Test_Active : BOOL;
    VO_Gas_Test_Active : BOOL;
    VO_Water_Test_Timeout_Close_Required : BOOL;
    VO_Gas_Test_Timeout_Close_Required : BOOL;
  END_VAR
  VAR
    L_CMD_Water_Selective_Recover_Prev : BOOL;
    L_CMD_Gas_Selective_Recover_Prev : BOOL;
    L_CMD_Water_Valve_Test_Open_Prev : BOOL;
    L_CMD_Water_Valve_Test_Close_Prev : BOOL;
    L_CMD_Water_Valve_Test_Confirm_Prev : BOOL;
    L_CMD_Gas_Valve_Test_Open_Prev : BOOL;
    L_CMD_Gas_Valve_Test_Close_Prev : BOOL;
    L_CMD_Gas_Valve_Test_Confirm_Prev : BOOL;
    L_Water_Test_Active : BOOL;
    L_Water_Test_Deadline : UDINT;
    L_Gas_Test_Active : BOOL;
    L_Gas_Test_Deadline : UDINT;
  END_VAR

            VO_Water_Test_Timeout_Close_Required := FALSE;
VO_Gas_Test_Timeout_Close_Required := FALSE;

VO_Water_Selective_Recover_Edge := VI_Water_Selective_Recover AND NOT L_CMD_Water_Selective_Recover_Prev;
VO_Gas_Selective_Recover_Edge := VI_Gas_Selective_Recover AND NOT L_CMD_Gas_Selective_Recover_Prev;
VO_Water_Valve_Test_Open_Edge := VI_Water_Valve_Test_Open AND NOT L_CMD_Water_Valve_Test_Open_Prev;
VO_Water_Valve_Test_Close_Edge := VI_Water_Valve_Test_Close AND NOT L_CMD_Water_Valve_Test_Close_Prev;
VO_Water_Valve_Test_Confirm_Edge := VI_Water_Valve_Test_Confirm AND NOT L_CMD_Water_Valve_Test_Confirm_Prev;
VO_Gas_Valve_Test_Open_Edge := VI_Gas_Valve_Test_Open AND NOT L_CMD_Gas_Valve_Test_Open_Prev;
VO_Gas_Valve_Test_Close_Edge := VI_Gas_Valve_Test_Close AND NOT L_CMD_Gas_Valve_Test_Close_Prev;
VO_Gas_Valve_Test_Confirm_Edge := VI_Gas_Valve_Test_Confirm AND NOT L_CMD_Gas_Valve_Test_Confirm_Prev;

L_CMD_Water_Selective_Recover_Prev := VI_Water_Selective_Recover;
L_CMD_Gas_Selective_Recover_Prev := VI_Gas_Selective_Recover;
L_CMD_Water_Valve_Test_Open_Prev := VI_Water_Valve_Test_Open;
L_CMD_Water_Valve_Test_Close_Prev := VI_Water_Valve_Test_Close;
L_CMD_Water_Valve_Test_Confirm_Prev := VI_Water_Valve_Test_Confirm;
L_CMD_Gas_Valve_Test_Open_Prev := VI_Gas_Valve_Test_Open;
L_CMD_Gas_Valve_Test_Close_Prev := VI_Gas_Valve_Test_Close;
L_CMD_Gas_Valve_Test_Confirm_Prev := VI_Gas_Valve_Test_Confirm;

IF VO_Water_Valve_Test_Open_Edge THEN
    L_Water_Test_Active := TRUE;
    L_Water_Test_Deadline := VI_System_Time_MS + 60000;
END_IF;

IF L_Water_Test_Active THEN
    IF VI_System_Time_MS >= L_Water_Test_Deadline THEN
        L_Water_Test_Active := FALSE;
        VO_Water_Test_Timeout_Close_Required := TRUE;
    END_IF;
END_IF;

IF VO_Gas_Valve_Test_Open_Edge THEN
    L_Gas_Test_Active := TRUE;
    L_Gas_Test_Deadline := VI_System_Time_MS + 60000;
END_IF;

IF L_Gas_Test_Active THEN
    IF VI_System_Time_MS >= L_Gas_Test_Deadline THEN
        L_Gas_Test_Active := FALSE;
        VO_Gas_Test_Timeout_Close_Required := TRUE;
    END_IF;
END_IF;

VO_Water_Test_Active := L_Water_Test_Active;
VO_Gas_Test_Active := L_Gas_Test_Active;
          
END_FUNCTION_BLOCK

FUNCTION_BLOCK FB_Smoke_Detector
  VAR_INPUT
    VI_Smoke_Signal : BOOL;
  END_VAR
  VAR_OUTPUT
    VO_Smoke_Detected : BOOL;
  END_VAR

            VO_Smoke_Detected := VI_Smoke_Signal;
          
END_FUNCTION_BLOCK

FUNCTION_BLOCK FB_System_Timebase
  VAR
    L_Time_Diff : UDINT;
  END_VAR

            // ==============================================================================
// System timebase helper
//
// Internal helper for PRG_System.
// Owns PLC runtime clock projection into GVL_STATUS:
// - monotonic system milliseconds
// - time-of-day milliseconds
// - day of week / day of year rollover
// - TOD representation
// ==============================================================================



GVL_STATUS.G_System_Time_MS := TIME_TO_UDINT(TIME());

L_Time_Diff := SEL(
    GVL_STATUS.G_System_Time_MS >= GVL_STATUS.G_Last_System_Time_MS,
    GVL_STATUS.G_System_Time_MS - GVL_STATUS.G_Last_System_Time_MS,
    (4294967295 - GVL_STATUS.G_Last_System_Time_MS) + GVL_STATUS.G_System_Time_MS + 1
);

GVL_STATUS.G_Time_Of_Day_MS := (GVL_STATUS.G_Time_Of_Day_MS + L_Time_Diff) MOD 86400000;

IF GVL_STATUS.G_Time_Of_Day_MS < L_Time_Diff THEN
    GVL_STATUS.G_Current_Day := (GVL_STATUS.G_Current_Day MOD 7) + 1;
    GVL_STATUS.G_Day_Of_Year := (GVL_STATUS.G_Day_Of_Year MOD 365) + 1;
END_IF;

GVL_STATUS.G_Last_System_Time_MS := GVL_STATUS.G_System_Time_MS;
GVL_STATUS.G_Current_TOD := UDINT_TO_TOD(GVL_STATUS.G_Time_Of_Day_MS);

// >>> BULK_SYNC_ANCHOR: FB_System_Timebase <<<
          
END_FUNCTION_BLOCK

FUNCTION_BLOCK FB_FloorHeating_Overheat_Protection
  VAR_INPUT
    VI_Threshold : REAL := 45.0;
  END_VAR
  VAR_OUTPUT
    VO_Overheat_Detected : BOOL;
    VO_Locked_Circuits : ARRAY[1..GVL_CONSTANTS.C_MAX_HEATING_CIRCUITS] OF BOOL;
  END_VAR
  VAR_IN_OUT
    VI_Temps : ARRAY[1..GVL_CONSTANTS.C_MAX_HEATING_CIRCUITS] OF REAL;
  END_VAR
  VAR
    L_i : INT;
  END_VAR

            VO_Overheat_Detected := FALSE;
FOR L_i := 1 TO GVL_CONSTANTS.C_MAX_HEATING_CIRCUITS DO
    IF VI_Temps[L_i] > VI_Threshold THEN
        VO_Overheat_Detected := TRUE;
        VO_Locked_Circuits[L_i] := TRUE;
    END_IF;
END_FOR;
          
END_FUNCTION_BLOCK

FUNCTION_BLOCK FB_CoreKernel_Live_Observer

            
          
END_FUNCTION_BLOCK

FUNCTION_BLOCK FB_LogEvent
  VAR_INPUT
    VI_Event_Type : UINT;
    VI_Timestamp : UDINT;
    VI_Param1 : UDINT;
    VI_Param2 : UDINT;
  END_VAR

            GVL_EVENT.G_Event_Log[GVL_EVENT.G_Event_Head].Event_ID := GVL_EVENT.G_Event_ID_Counter;
GVL_EVENT.G_Event_Log[GVL_EVENT.G_Event_Head].Event_Type := VI_Event_Type;
GVL_EVENT.G_Event_Log[GVL_EVENT.G_Event_Head].Timestamp := VI_Timestamp;
GVL_EVENT.G_Event_Log[GVL_EVENT.G_Event_Head].Param1 := VI_Param1;
GVL_EVENT.G_Event_Log[GVL_EVENT.G_Event_Head].Param2 := VI_Param2;

GVL_EVENT.G_Event_ID_Counter := GVL_EVENT.G_Event_ID_Counter + 1;
GVL_EVENT.G_Event_Head := (GVL_EVENT.G_Event_Head + 1) MOD 64;
          
END_FUNCTION_BLOCK

FUNCTION_BLOCK FB_System_Gateway_Intent
  VAR_INPUT
    VI_System_Time_MS : UDINT;
    VI_IsActivePLC : BOOL;
    VI_Gateway_Writes_Allowed : BOOL;
  END_VAR
  VAR_IN_OUT
    VIO_FloorHeating_Temps : ARRAY[1..8] OF REAL;
    VIO_Zone_Valve_States : ARRAY[1..8] OF BOOL;
    VIO_Lighting_Base_Levels : ARRAY[1..32] OF BYTE;
    VIO_Scenario_Req_Gateway : E_SCENARIO_TYPE;
  END_VAR
  VAR
    fbGateway : FB_Gateway_Interface;
  END_VAR

            // ==============================================================================
// System gateway intent helper
//
// Internal helper for PRG_System.
// Owns gateway FB call, user intent publication, gateway command gates,
// and allowed configuration/time/scenario writes.
// ==============================================================================



fbGateway(
    VI_System_Time_MS := VI_System_Time_MS,
    VI_Local_PLC_Role := SEL(VI_IsActivePLC, E_PLC_ROLE.ROLE_STANDBY, E_PLC_ROLE.ROLE_ACTIVE),
    VI_Incoming_Command := GVL_GATEWAY.G_Gateway_Command,
    VI_Command_Received := GVL_GATEWAY.G_Gateway_Command_Received,
    VI_FloorHeating_Temps := VIO_FloorHeating_Temps,
    VI_Room_Temps := GVL_STATE.G_Room_Temps,
    VI_Zone_Valve_States := VIO_Zone_Valve_States,
    VI_Manifold_Pressures := GVL_STATE.G_Manifold_Pressures,
    VI_Manifold_Pump_States := GVL_STATE.G_Manifold_Pumps,
    VI_Outdoor_Temp := GVL_STATE.G_Outdoor_Temp,
    VI_Security_Armed := GVL_ALARM.G_Security_Armed,
    VI_Flood_Alarm_Active := GVL_ALARM.G_Flood_Alarm_Active,
    VI_Gas_Alarm_Active := GVL_ALARM.G_Gas_Alarm_Active,
    VI_Fire_Alarm_Active := GVL_ALARM.G_Fire_Alarm_Active,
    VI_Methane_Concentration := GVL_STATE.G_Methane_Sensors[1],
    VI_Lighting_Base_Levels := VIO_Lighting_Base_Levels,
    VI_Socket_States := GVL_STATE.G_Socket_States,
    VI_Blinds_Positions := GVL_STATE.G_Blinds_Positions,
    VI_Active_Scenario := GVL_STATUS.G_Current_Scenario,
    VI_Send_2FA_Req := GVL_COMMAND.G_Send_2FA_Req,
    VI_2FA_Code := GVL_COMMAND.G_2FA_Code_Out,
    VI_Allowed_IPs := GVL_CONFIG.G_Allowed_IPs,
    VO_Telegram_Msg => GVL_GATEWAY.G_Gateway_Telegram_Msg,
    VO_Send_Telegram => GVL_GATEWAY.G_Gateway_Send_Telegram,
    VO_HMI_Status_Message => GVL_GATEWAY.G_Gateway_HMI_Status_Message,

    VO_Data_Ready => GVL_GATEWAY.G_Gateway_Data_Ready,
    VO_Modbus_Registers => GVL_GATEWAY.G_Gateway_Modbus_Registers,
    VO_Arm_Req => GVL_COMMAND.G_Arm_Req,
    VO_Disarm_Req => GVL_COMMAND.G_Disarm_Req,
    VO_PIN_Code => GVL_COMMAND.G_PIN_Code,
    VO_RFID_Tag => GVL_COMMAND.G_RFID_Tag,
    VO_2FA_Code_In => GVL_COMMAND.G_2FA_Code_In,
    VO_Lighting_Override => GVL_COMMAND.G_Lighting_Override,
    VO_Blinds_Override => GVL_COMMAND.G_Blinds_Override,
    VO_Socket_Override => GVL_COMMAND.G_Socket_Override,
    VO_Reset_Errors_Req => GVL_COMMAND.G_Reset_Errors
);

GVL_INTENT_USER.I_Source_Valid := TRUE;
GVL_INTENT_USER.I_Last_Update_MS := VI_System_Time_MS;
GVL_INTENT_USER.I_Arm_Request := GVL_COMMAND.G_Arm_Req;
GVL_INTENT_USER.I_Disarm_Request := GVL_COMMAND.G_Disarm_Req;
GVL_INTENT_USER.I_PIN_Code := GVL_COMMAND.G_PIN_Code;
GVL_INTENT_USER.I_RFID_Tag := GVL_COMMAND.G_RFID_Tag;
GVL_INTENT_USER.I_2FA_Code_In := GVL_COMMAND.G_2FA_Code_In;
GVL_INTENT_USER.I_Lighting_Override_32 := GVL_COMMAND.G_Lighting_Override;
GVL_INTENT_USER.I_Blinds_Override_32 := GVL_COMMAND.G_Blinds_Override;
GVL_INTENT_USER.I_Socket_Override_32 := GVL_COMMAND.G_Socket_Override;
GVL_INTENT_USER.I_Reset_Errors := GVL_COMMAND.G_Reset_Errors;
GVL_INTENT_USER.I_Set_Temp_Req := fbGateway.VO_Set_Temp_Req;
GVL_INTENT_USER.I_Target_Zone := fbGateway.VO_Target_Zone;
GVL_INTENT_USER.I_Target_Temperature := fbGateway.VO_Target_Temp;
GVL_INTENT_USER.I_Set_Vent_Req := fbGateway.VO_Set_Vent_Req;
GVL_INTENT_USER.I_Target_Vent_Speed := fbGateway.VO_Target_Vent_Speed;
GVL_INTENT_USER.I_Set_Config_Req := fbGateway.VO_Set_Config_Req;
GVL_INTENT_USER.I_Time_Sync_Req := fbGateway.VO_Sync_Time_Req;
GVL_INTENT_USER.I_New_Time_MS := fbGateway.VO_New_Time_MS;

IF VI_Gateway_Writes_Allowed AND
   fbGateway.VO_Set_Scenario_Req AND
   ((GVL_STATE.G_System_Mode = E_System_Operating_Mode.MODE_NORMAL) OR
    (GVL_STATE.G_System_Mode = E_System_Operating_Mode.MODE_DEGRADED)) THEN
    VIO_Scenario_Req_Gateway := fbGateway.VO_Target_Scenario;
END_IF;

IF VI_Gateway_Writes_Allowed AND
   fbGateway.VO_Set_Temp_Req AND
   (GVL_STATE.G_System_Mode = E_System_Operating_Mode.MODE_NORMAL) THEN
    GVL_CONFIG.G_HMI_FloorHeating_Configs[fbGateway.VO_Target_Zone].design_temp := fbGateway.VO_Target_Temp;
END_IF;

IF VI_Gateway_Writes_Allowed AND
   fbGateway.VO_Set_Vent_Req AND
   (GVL_STATE.G_System_Mode = E_System_Operating_Mode.MODE_NORMAL) THEN
    GVL_CONFIG.G_HMI_Vent_Global_Config.default_supply_speed := fbGateway.VO_Target_Vent_Speed;
END_IF;

IF VI_Gateway_Writes_Allowed AND
   fbGateway.VO_Set_Config_Req AND
   (GVL_STATE.G_System_Mode = E_System_Operating_Mode.MODE_NORMAL) THEN
    GVL_CONFIG.G_HMI_Apply_Settings := TRUE;
END_IF;

IF VI_Gateway_Writes_Allowed AND
   fbGateway.VO_Sync_Time_Req AND
   (GVL_STATE.G_System_Mode = E_System_Operating_Mode.MODE_NORMAL) THEN
    GVL_STATUS.G_Time_Of_Day_MS := fbGateway.VO_New_Time_MS;
END_IF;

GVL_INTENT_USER.I_Scenario_Request := VIO_Scenario_Req_Gateway;
GVL_INTENT_USER.I_Gate_Open_Request := GVL_COMMAND.G_Gate_Open;
GVL_INTENT_USER.I_Wicket_Open_Request := GVL_COMMAND.G_Wicket_Open;
GVL_INTENT_USER.I_Lock_1_Open_Request := GVL_COMMAND.G_Lock_1_Open;
GVL_INTENT_USER.I_Lock_1_Close_Request := GVL_COMMAND.G_Lock_1_Close;
GVL_INTENT_USER.I_Lock_2_Open_Request := GVL_COMMAND.G_Lock_2_Open;
GVL_INTENT_USER.I_Lock_2_Close_Request := GVL_COMMAND.G_Lock_2_Close;
GVL_INTENT_USER.I_Dangerous_Action_Request := GVL_COMMAND.CMD_Dangerous_Action_Request;
GVL_INTENT_USER.I_Dangerous_Action_Confirm := GVL_COMMAND.CMD_Dangerous_Action_Confirm;
GVL_INTENT_USER.I_User_Access_Level := GVL_COMMAND.CMD_User_Access_Level;
GVL_INTENT_USER.I_Water_Selective_Recover := GVL_COMMAND.CMD_Water_Selective_Recover;
GVL_INTENT_USER.I_Gas_Selective_Recover := GVL_COMMAND.CMD_Gas_Selective_Recover;

// >>> BULK_SYNC_ANCHOR: FB_System_Gateway_Intent <<<
          
END_FUNCTION_BLOCK

FUNCTION_BLOCK FB_Redundancy_Manager
  VAR_INPUT
    VI_System_Time_MS : UDINT;
    VI_Local_PLC_ID : BYTE;
    VI_Remote_Pulse : BOOL;
    VI_Remote_Is_Active : BOOL;
    VI_Gateway_Ping_OK : BOOL;
    VI_Remote_State : ST_System_State_Snapshot;
    VI_Local_State : ST_System_State_Snapshot;
  END_VAR
  VAR_OUTPUT
    VO_Local_Role : E_PLC_ROLE;
    VO_Local_Pulse : BOOL;
    VO_Sync_Data_Req : BOOL;
    VO_Status_Msg : STRING(200);
    VO_Synced_State : ST_System_State_Snapshot;
    VO_State_Updated : BOOL;
  END_VAR
  VAR
    L_Heartbeat : FB_PLC_Heartbeat;
    L_Pulse_Timer : FB_System_Timer;
    L_Pulse_State : BOOL;
    L_Prev_Role : E_PLC_ROLE;
    L_State_Replicator : FB_State_Replication;
  END_VAR

            // 1. Генерация собственного пульса (меандр 100 мс)
L_Pulse_Timer(IN := NOT L_Pulse_Timer.Q, PT := T#100ms, VI_System_Time_MS := VI_System_Time_MS);
IF L_Pulse_Timer.Q THEN
    L_Pulse_State := NOT L_Pulse_State;
END_IF;
VO_Local_Pulse := L_Pulse_State;

// 2. Определение роли через Heartbeat
L_Heartbeat(
    VI_Local_ID := VI_Local_PLC_ID,
    VI_System_Time := VI_System_Time_MS,
    VI_Remote_Pulse := VI_Remote_Pulse,
    VI_Remote_Is_Active := VI_Remote_Is_Active,
    VI_Gateway_Ping_OK := VI_Gateway_Ping_OK
);

IF L_Heartbeat.VO_Is_Active THEN
    VO_Local_Role := E_PLC_ROLE.ROLE_ACTIVE;
    VO_Status_Msg := 'ПЛК АКТИВЕН (ВЕДУЩИЙ)';
ELSE
    VO_Local_Role := E_PLC_ROLE.ROLE_STANDBY;
    VO_Status_Msg := 'ПЛК В РЕЗЕРВЕ (ВЕДОМЫЙ)';
END_IF;

// 3. Запрос на синхронизацию при переходе в ACTIVE
IF VO_Local_Role = E_PLC_ROLE.ROLE_ACTIVE AND L_Prev_Role = E_PLC_ROLE.ROLE_STANDBY THEN
    VO_Sync_Data_Req := TRUE;
ELSE
    VO_Sync_Data_Req := FALSE;
END_IF;

L_State_Replicator(
    VI_Local_Role := VO_Local_Role,
    VI_Sync_Req := VO_Sync_Data_Req,
    VI_Local_State := VI_Local_State,
    VI_Remote_State := VI_Remote_State,
    VI_System_Time_MS := VI_System_Time_MS
);
VO_Synced_State := L_State_Replicator.VO_Synced_State;
VO_State_Updated := L_State_Replicator.VO_State_Updated;

L_Prev_Role := VO_Local_Role;
// >>> BULK_SYNC_ANCHOR: FB_Redundancy_Manager <<<
          
END_FUNCTION_BLOCK

FUNCTION_BLOCK FB_Security_System_Manager
  VAR_INPUT
    VI_System_Time_MS : UDINT;
    VI_IsActivePLC : BOOL;
    VI_Arm_Request : BOOL;
    VI_Disarm_Request : BOOL;
    VI_PIN_Code : STRING(4);
    VI_RFID_Tag : STRING(20);
    VI_2FA_Code : STRING(6);
    VI_Config : ST_Security_Global_Config;
    VI_Current_TOD : TOD;
  END_VAR
  VAR_OUTPUT
    VO_Armed : BOOL;
    VO_Alarm_Active : BOOL;
    VO_Siren_Active : BOOL;
    VO_Status_Msg : STRING(200);
    VO_Send_Code_Req : BOOL;
    VO_Code_To_Send : STRING(6);
  END_VAR
  VAR_IN_OUT
    VI_Motion_Sensors : ARRAY[1..16] OF BOOL;
    VI_Door_Sensors : ARRAY[1..GVL_CONSTANTS.C_MAX_DOOR_SENSORS] OF BOOL;
    VI_Window_Sensors : ARRAY[1..16] OF BOOL;
    VI_Bypass_Motion : ARRAY[1..16] OF BOOL;
    VI_Bypass_Doors : ARRAY[1..GVL_CONSTANTS.C_MAX_DOOR_SENSORS] OF BOOL;
    VI_Bypass_Windows : ARRAY[1..16] OF BOOL;
  END_VAR
  VAR
    L_i : INT;
    L_Any_Sensor_Active : BOOL;
    L_Arm_Delay_Timer : FB_System_Timer;
    L_Alarm_Delay_Timer : FB_System_Timer;
    L_Arming_In_Progress : BOOL;
    L_Valid_PIN : BOOL;
    fbAccessCode : FB_AccessCode_Manager;
    fbTwoFactor : FB_TwoFactor_Auth;
    L_2FA_Required : BOOL;
    L_Disarm_Pending : BOOL;
    L_Reset_2FA : BOOL;
    L_Auto_Arm_Trigger : BOOL;
    R_Trig_Auto_Arm : R_TRIG;
  END_VAR

            IF NOT VI_IsActivePLC THEN
    VO_Armed := FALSE;
    VO_Alarm_Active := FALSE;
    VO_Siren_Active := FALSE;
    VO_Send_Code_Req := FALSE;
    VO_Code_To_Send := '';
    VO_Status_Msg := 'Охрана: резервный ПЛК';
    L_Arming_In_Progress := FALSE;
    L_Disarm_Pending := FALSE;
    L_2FA_Required := FALSE;
    L_Reset_2FA := FALSE;
    RETURN;
END_IF;

// 1. Проверка PIN-кода или RFID-метки через менеджер кодов
fbAccessCode(
    VI_System_Time_MS := VI_System_Time_MS,
    VI_IsActivePLC := VI_IsActivePLC,
    VI_Code_To_Check := VI_PIN_Code,
    VI_RFID_To_Check := VI_RFID_Tag,
    VI_Access_Codes := GVL_RETAIN.G_Access_Codes,
    VI_RFID_Tags := GVL_RETAIN.G_RFID_Tags,
    VO_Code_Valid => L_Valid_PIN
);

// 2. Логика постановки на охрану (с задержкой на выход)
L_Auto_Arm_Trigger := FALSE;
IF VI_Config.auto_arm_enabled THEN
    IF VI_Current_TOD >= UDINT_TO_TOD(VI_Config.auto_arm_time_ms) THEN
        L_Auto_Arm_Trigger := TRUE;
    END_IF;
END_IF;
R_Trig_Auto_Arm(CLK := L_Auto_Arm_Trigger);

IF ((VI_Arm_Request AND L_Valid_PIN) OR R_Trig_Auto_Arm.Q) AND NOT VO_Armed AND NOT L_Arming_In_Progress THEN
    // Проверка, что все двери/окна закрыты перед постановкой (с учетом байпаса)
    L_Any_Sensor_Active := FALSE;
    FOR L_i := 1 TO GVL_CONSTANTS.C_MAX_DOOR_SENSORS DO IF VI_Door_Sensors[L_i] AND NOT VI_Bypass_Doors[L_i] THEN L_Any_Sensor_Active := TRUE; END_IF; END_FOR;
    FOR L_i := 1 TO 16 DO IF VI_Window_Sensors[L_i] AND NOT VI_Bypass_Windows[L_i] THEN L_Any_Sensor_Active := TRUE; END_IF; END_FOR;
    
    IF NOT L_Any_Sensor_Active THEN
        L_Arming_In_Progress := TRUE;
        VO_Status_Msg := 'Постановка на охрану. Покиньте помещение.';
    ELSE
        VO_Status_Msg := 'Ошибка постановки: Открыты двери или окна';
    END_IF;
END_IF;

L_Arm_Delay_Timer(IN := L_Arming_In_Progress, PT := TO_TIME(VI_Config.exit_delay_seconds * 1000), VI_System_Time_MS := VI_System_Time_MS);
IF L_Arm_Delay_Timer.Q THEN
    L_Arming_In_Progress := FALSE;
    VO_Armed := TRUE;
    VO_Status_Msg := 'Система под охраной';
END_IF;

// 3. Логика снятия с охраны с 2FA
IF VI_Disarm_Request AND L_Valid_PIN AND VO_Armed THEN
    IF VI_Config.enable_2fa THEN
        L_Disarm_Pending := TRUE;
        L_2FA_Required := TRUE;
        VO_Status_Msg := 'Ожидание 2FA для снятия с охраны';
    ELSE
        // Снятие без 2FA
        VO_Armed := FALSE;
        VO_Alarm_Active := FALSE;
        VO_Siren_Active := FALSE;
        L_Arming_In_Progress := FALSE;
        VO_Status_Msg := 'Система снята с охраны';
    END_IF;
END_IF;

fbTwoFactor(
    VI_System_Time_MS := VI_System_Time_MS,
    VI_Start_Auth := L_2FA_Required,
    VI_Method := E_TwoFactor_Method.TF_METHOD_TOTP, // Для примера
    VI_User_Code := VI_2FA_Code, // Используем отдельный вход для 2FA кода
    VI_Reset_Success := L_Reset_2FA
);

VO_Send_Code_Req := fbTwoFactor.VO_Send_Code_Req;
VO_Code_To_Send := fbTwoFactor.VO_Code_To_Send;

IF L_Disarm_Pending AND fbTwoFactor.VO_State.Is_Success THEN
    VO_Armed := FALSE;
    VO_Alarm_Active := FALSE;
    VO_Siren_Active := FALSE;
    L_Arming_In_Progress := FALSE;
    L_Disarm_Pending := FALSE;
    L_2FA_Required := FALSE;
    L_Reset_2FA := TRUE;
    VO_Status_Msg := 'Система снята с охраны';
ELSIF L_Disarm_Pending AND fbTwoFactor.VO_State.Is_Locked THEN
    L_Disarm_Pending := FALSE;
    L_2FA_Required := FALSE;
    L_Reset_2FA := FALSE;
    VO_Status_Msg := 'Ошибка 2FA: Превышено количество попыток';
ELSE
    L_Reset_2FA := FALSE;
END_IF;

// 4. Логика тревоги (с задержкой на вход)
IF VO_Armed THEN
    L_Any_Sensor_Active := FALSE;
    FOR L_i := 1 TO 16 DO IF VI_Motion_Sensors[L_i] AND NOT VI_Bypass_Motion[L_i] THEN L_Any_Sensor_Active := TRUE; END_IF; END_FOR;
    FOR L_i := 1 TO GVL_CONSTANTS.C_MAX_DOOR_SENSORS DO IF VI_Door_Sensors[L_i] AND NOT VI_Bypass_Doors[L_i] THEN L_Any_Sensor_Active := TRUE; END_IF; END_FOR;
    FOR L_i := 1 TO 16 DO IF VI_Window_Sensors[L_i] AND NOT VI_Bypass_Windows[L_i] THEN L_Any_Sensor_Active := TRUE; END_IF; END_FOR;
    
    // Защелкиваем факт нарушения периметра, чтобы кратковременное срабатывание датчика не сбрасывало таймер
    IF L_Any_Sensor_Active THEN
        L_Alarm_Delay_Timer.IN := TRUE;
    END_IF;
    
    L_Alarm_Delay_Timer(PT := TO_TIME(VI_Config.entry_delay_seconds * 1000), VI_System_Time_MS := VI_System_Time_MS);
    
    IF L_Alarm_Delay_Timer.Q THEN
        VO_Alarm_Active := TRUE;
        VO_Siren_Active := TRUE;
        VO_Status_Msg := 'ТРЕВОГА! Нарушение периметра';
    ELSIF L_Alarm_Delay_Timer.IN THEN
        VO_Status_Msg := 'Внимание! Введите PIN-код для отмены тревоги';
    END_IF;
ELSE
    L_Alarm_Delay_Timer(IN := FALSE, PT := T#0s, VI_System_Time_MS := VI_System_Time_MS); // Сброс таймера при снятии с охраны
END_IF;
// >>> BULK_SYNC_ANCHOR: FB_Security_System_Manager <<<
          
END_FUNCTION_BLOCK

FUNCTION_BLOCK FB_Rule_Engine
  VAR_INPUT
    VI_System_Time_MS : UDINT;
    VI_IsActivePLC : BOOL;
    VI_Security_Armed : BOOL;
    VI_Current_Time : TOD;
    VI_Day_Of_Week : INT;
  END_VAR
  VAR_OUTPUT
    VO_Preheat_Request : BOOL;
    VO_Actions : ARRAY[1..GVL_CONSTANTS.C_MAX_RULES] OF ST_Rule_Action;
  END_VAR
  VAR_IN_OUT
    VI_Rules : ARRAY[1..GVL_CONSTANTS.C_MAX_RULES] OF ST_User_Rule;
    VI_Indoor_Temps : ARRAY[1..16] OF REAL;
    VI_Floor_Temps : ARRAY[1..8] OF REAL;
    VI_Humidities : ARRAY[1..16] OF REAL;
    VI_CO2_Levels : ARRAY[1..16] OF REAL;
    VI_Motion_Sensors : ARRAY[1..16] OF BOOL;
    VI_Door_Sensors : ARRAY[1..GVL_CONSTANTS.C_MAX_DOOR_SENSORS] OF BOOL;
    VI_Window_Sensors : ARRAY[1..16] OF BOOL;
    VI_Water_Sensors : ARRAY[1..GVL_CONSTANTS.C_MAX_FLOOD_SENSORS] OF BOOL;
    VI_Smoke_Sensors : ARRAY[1..GVL_CONSTANTS.C_MAX_SMOKE_SENSORS] OF BOOL;
    VI_Methane_Sensors : ARRAY[1..GVL_CONSTANTS.C_MAX_METHANE_SENSORS] OF REAL;
    VI_CO_Sensors : ARRAY[1..GVL_CONSTANTS.C_MAX_CO_SENSORS] OF REAL;
  END_VAR
  VAR
    L_i : INT;
    L_Condition_Met : BOOL;
    L_Current_Value : REAL;
    L_Triggers : ARRAY[1..GVL_CONSTANTS.C_MAX_RULES] OF R_TRIG;
    L_Trigger_Count : ARRAY[1..GVL_CONSTANTS.C_MAX_RULES] OF UINT;
    L_Last_Reset_Time : UDINT;
    L_Elapsed_Time : UDINT;
  END_VAR

            IF NOT VI_IsActivePLC THEN RETURN; END_IF;

VO_Preheat_Request := FALSE;


// Сброс счетчиков срабатываний каждую минуту (защита от циклических зависимостей/дребезга)
L_Elapsed_Time := (SEL(VI_System_Time_MS >= L_Last_Reset_Time, VI_System_Time_MS - L_Last_Reset_Time, (4294967295 - L_Last_Reset_Time) + VI_System_Time_MS + 1));

IF L_Elapsed_Time >= GVL_CONSTANTS.C_MS_IN_MINUTE THEN
    L_Last_Reset_Time := VI_System_Time_MS;
    FOR L_i := 1 TO GVL_CONSTANTS.C_MAX_RULES DO
        L_Trigger_Count[L_i] := 0;
    END_FOR;
END_IF;

FOR L_i := 1 TO GVL_CONSTANTS.C_MAX_RULES DO

    VO_Actions[L_i].Active := FALSE;
    IF VI_Rules[L_i].Enabled THEN
        L_Condition_Met := FALSE;
        L_Current_Value := 0.0;
        
        // Определение значения для проверки
        IF VI_Rules[L_i].Condition_Target_ID > 0 THEN
            CASE VI_Rules[L_i].Condition_Type OF
                E_Rule_Condition_Type.COND_AIR_TEMP: IF VI_Rules[L_i].Condition_Target_ID <= 16 THEN L_Current_Value := VI_Indoor_Temps[VI_Rules[L_i].Condition_Target_ID]; END_IF;
                E_Rule_Condition_Type.COND_FLOOR_TEMP: IF VI_Rules[L_i].Condition_Target_ID <= 8 THEN L_Current_Value := VI_Floor_Temps[VI_Rules[L_i].Condition_Target_ID]; END_IF;
                E_Rule_Condition_Type.COND_HUMIDITY: IF VI_Rules[L_i].Condition_Target_ID <= 16 THEN L_Current_Value := VI_Humidities[VI_Rules[L_i].Condition_Target_ID]; END_IF;
                E_Rule_Condition_Type.COND_CO2: IF VI_Rules[L_i].Condition_Target_ID <= 16 THEN L_Current_Value := VI_CO2_Levels[VI_Rules[L_i].Condition_Target_ID]; END_IF;
                E_Rule_Condition_Type.COND_MOTION: IF VI_Rules[L_i].Condition_Target_ID <= 16 THEN L_Current_Value := SEL(VI_Motion_Sensors[VI_Rules[L_i].Condition_Target_ID], 0.0, 1.0); END_IF;
                E_Rule_Condition_Type.COND_DOOR_WINDOW: 
                    IF VI_Rules[L_i].Condition_Target_ID <= GVL_CONSTANTS.C_MAX_DOOR_SENSORS THEN
                        L_Current_Value := SEL(VI_Door_Sensors[VI_Rules[L_i].Condition_Target_ID] OR VI_Window_Sensors[VI_Rules[L_i].Condition_Target_ID], 0.0, 1.0);
                    ELSIF VI_Rules[L_i].Condition_Target_ID <= 16 THEN
                        L_Current_Value := SEL(VI_Window_Sensors[VI_Rules[L_i].Condition_Target_ID], 0.0, 1.0);
                    END_IF;
                E_Rule_Condition_Type.COND_FLOOD: IF VI_Rules[L_i].Condition_Target_ID <= GVL_CONSTANTS.C_MAX_FLOOD_SENSORS THEN L_Current_Value := SEL(VI_Water_Sensors[VI_Rules[L_i].Condition_Target_ID], 0.0, 1.0); END_IF;
                E_Rule_Condition_Type.COND_SMOKE: IF VI_Rules[L_i].Condition_Target_ID <= GVL_CONSTANTS.C_MAX_SMOKE_SENSORS THEN L_Current_Value := SEL(VI_Smoke_Sensors[VI_Rules[L_i].Condition_Target_ID], 0.0, 1.0); END_IF;
                E_Rule_Condition_Type.COND_METHANE: IF VI_Rules[L_i].Condition_Target_ID <= GVL_CONSTANTS.C_MAX_METHANE_SENSORS THEN L_Current_Value := VI_Methane_Sensors[VI_Rules[L_i].Condition_Target_ID]; END_IF;
                E_Rule_Condition_Type.COND_CO: IF VI_Rules[L_i].Condition_Target_ID <= GVL_CONSTANTS.C_MAX_CO_SENSORS THEN L_Current_Value := VI_CO_Sensors[VI_Rules[L_i].Condition_Target_ID]; END_IF;
                E_Rule_Condition_Type.COND_TIME_OF_DAY: L_Current_Value := TO_REAL(TOD_TO_UDINT(VI_Current_Time) / GVL_CONSTANTS.C_MS_IN_MINUTE); // Время в минутах
                E_Rule_Condition_Type.COND_DAY_OF_WEEK: L_Current_Value := TO_REAL(VI_Day_Of_Week);
            END_CASE;
        ELSE
            IF VI_Rules[L_i].Condition_Type = E_Rule_Condition_Type.COND_TIME_OF_DAY THEN
                L_Current_Value := TO_REAL(TOD_TO_UDINT(VI_Current_Time) / GVL_CONSTANTS.C_MS_IN_MINUTE); // Время в минутах
            ELSIF VI_Rules[L_i].Condition_Type = E_Rule_Condition_Type.COND_DAY_OF_WEEK THEN
                L_Current_Value := TO_REAL(VI_Day_Of_Week);
            END_IF;
        END_IF;
        
        // Проверка условия
        CASE VI_Rules[L_i].Condition_Op OF
            E_Rule_Comparison.COMP_GT: L_Condition_Met := (L_Current_Value > VI_Rules[L_i].Condition_Value);
            E_Rule_Comparison.COMP_LT: L_Condition_Met := (L_Current_Value < VI_Rules[L_i].Condition_Value);
            E_Rule_Comparison.COMP_EQ: L_Condition_Met := (ABS(L_Current_Value - VI_Rules[L_i].Condition_Value) < 0.1);
            E_Rule_Comparison.COMP_GE: L_Condition_Met := (L_Current_Value >= VI_Rules[L_i].Condition_Value);
            E_Rule_Comparison.COMP_LE: L_Condition_Met := (L_Current_Value <= VI_Rules[L_i].Condition_Value);
            E_Rule_Comparison.COMP_IN_RANGE: L_Condition_Met := (L_Current_Value >= VI_Rules[L_i].Condition_Value) AND (L_Current_Value <= VI_Rules[L_i].Condition_Value_Max);
            E_Rule_Comparison.COMP_TRUE: L_Condition_Met := (L_Current_Value > 0.5);
            E_Rule_Comparison.COMP_FALSE: L_Condition_Met := (L_Current_Value < 0.5);
        END_CASE;
        
        // Формирование действия
        L_Triggers[L_i](CLK := L_Condition_Met);
        
        IF L_Triggers[L_i].Q THEN
            L_Trigger_Count[L_i] := L_Trigger_Count[L_i] + 1;
            IF L_Trigger_Count[L_i] > 10 THEN
                // ТЗ 13.5: Блокировка правила при слишком частом срабатывании (циклическая зависимость)
                VO_Actions[L_i].Active := FALSE;
                VO_Actions[L_i].Triggered := FALSE;
                CONTINUE; // Пропускаем выполнение
            END_IF;
        END_IF;
        
        IF L_Condition_Met AND (L_Trigger_Count[L_i] <= 10) THEN
            VO_Actions[L_i].Active := TRUE;
            VO_Actions[L_i].Triggered := L_Triggers[L_i].Q;
            VO_Actions[L_i].Action_Type := VI_Rules[L_i].Action_Type;
            VO_Actions[L_i].Target_ID := VI_Rules[L_i].Action_Target_ID;
            VO_Actions[L_i].Value := VI_Rules[L_i].Action_Value;
        END_IF;
    END_IF;
END_FOR;
// >>> BULK_SYNC_ANCHOR: FB_Rule_Engine <<<
          
END_FUNCTION_BLOCK

FUNCTION_BLOCK FB_Heating_Safety_Gate
  VAR_INPUT
    VI_System_Mode : E_System_Operating_Mode;
    VI_Emergency_Stop : BOOL;
    VI_Gas_Safety_Stop : BOOL;
    VI_IO_Failsafe_Active : BOOL;
    VI_Outdoor_Temp : REAL;
    VI_Freeze_Threshold : REAL;
  END_VAR
  VAR_OUTPUT
    VO_Block_Normal_Heating : BOOL;
    VO_Gas_Safety_Active : BOOL;
    VO_Emergency_Safe_Stop_Active : BOOL;
    VO_IO_Failsafe_Active : BOOL;
    VO_Freeze_Mode_Active : BOOL;
    VO_Freeze_Target_Supply : REAL;
  END_VAR
  VAR_IN_OUT
    VI_Floor_Temps : ARRAY[1..GVL_CONSTANTS.C_MAX_HEATING_CIRCUITS] OF REAL;
  END_VAR
  VAR
    L_i : INT;
  END_VAR

            // ==============================================================================
// Heating safety gate helper
//
// Internal helper for FB_Heating_System_Manager.
// Owns common safety/freeze decision calculation. The manager remains the public
// facade and still projects physical safe-state outputs.
// ==============================================================================



VO_Gas_Safety_Active := VI_Gas_Safety_Stop;
VO_Emergency_Safe_Stop_Active := VI_Emergency_Stop OR (VI_System_Mode = E_System_Operating_Mode.MODE_SAFE_STOP);
VO_IO_Failsafe_Active := VI_IO_Failsafe_Active;

VO_Block_Normal_Heating := VO_Gas_Safety_Active OR VO_Emergency_Safe_Stop_Active OR VO_IO_Failsafe_Active;
VO_Freeze_Mode_Active := (VI_System_Mode = E_System_Operating_Mode.MODE_FREEZE_PROTECTION) OR (VI_Outdoor_Temp < -5.0);

FOR L_i := 1 TO GVL_CONSTANTS.C_MAX_HEATING_CIRCUITS DO
    IF VI_Floor_Temps[L_i] < 7.0 THEN
        VO_Freeze_Mode_Active := TRUE;
    END_IF;
END_FOR;

IF VO_Freeze_Mode_Active THEN
    VO_Freeze_Target_Supply := LIMIT(20.0, VI_Freeze_Threshold + 2.0, 35.0);
ELSE
    VO_Freeze_Target_Supply := 0.0;
END_IF;

// >>> BULK_SYNC_ANCHOR: FB_Heating_Safety_Gate <<<
          
END_FUNCTION_BLOCK

FUNCTION_BLOCK FB_Lifetime_Manager
  VAR_INPUT
    VI_System_Time_MS : UDINT;
    VI_Device_Active : BOOL;
    VI_Device_ID : BYTE;
    VI_Nominal_Hours : UDINT;
  END_VAR
  VAR_IN_OUT
    VIO_Status : ST_Lifetime_Status;
  END_VAR
  VAR
    L_Last_Time : UDINT;
    L_Prev_State : BOOL;
    L_Delta_MS : UDINT;
    L_Runtime_Accum_MS : UDINT;
    L_Remaining_Percent_UDINT : UDINT;
  END_VAR

            // === DELTA TIME ===
IF VI_System_Time_MS >= L_Last_Time THEN
    L_Delta_MS := VI_System_Time_MS - L_Last_Time;
ELSE
    // overflow
    L_Delta_MS := (4294967295 - L_Last_Time) + VI_System_Time_MS + 1;
END_IF;

L_Last_Time := VI_System_Time_MS;

// === START COUNT ===
IF VI_Device_Active AND NOT L_Prev_State THEN
    VIO_Status.start_count := VIO_Status.start_count + 1;
END_IF;

L_Prev_State := VI_Device_Active;

// === RUNTIME ACCUMULATION ===
IF VI_Device_Active THEN
    L_Runtime_Accum_MS := L_Runtime_Accum_MS + L_Delta_MS;

    WHILE L_Runtime_Accum_MS >= 3600000 DO
        VIO_Status.runtime_hours := VIO_Status.runtime_hours + 1;
        L_Runtime_Accum_MS := L_Runtime_Accum_MS - 3600000;
    END_WHILE;
END_IF;

// === BASIC LIFETIME ESTIMATION ===
IF VI_Nominal_Hours > 0 THEN
    IF VIO_Status.runtime_hours >= VI_Nominal_Hours THEN
        VIO_Status.remaining_hours := 0;
        VIO_Status.remaining_percent := 0;
    ELSE
        VIO_Status.remaining_hours := VI_Nominal_Hours - VIO_Status.runtime_hours;
        L_Remaining_Percent_UDINT := (VIO_Status.remaining_hours * 100) / VI_Nominal_Hours;

        IF L_Remaining_Percent_UDINT > 100 THEN
            L_Remaining_Percent_UDINT := 100;
        END_IF;

        VIO_Status.remaining_percent := UDINT_TO_BYTE(L_Remaining_Percent_UDINT);
    END_IF;
ELSE
    VIO_Status.remaining_hours := 0;
    VIO_Status.remaining_percent := 0;
END_IF;

VIO_Status.maintenance_required := VIO_Status.remaining_percent <= GVL_Lifetime.G_Maintenance_Threshold_Percent;

// === BASIC FLAGS ===
VIO_Status.device_id := VI_Device_ID;
VIO_Status.last_calc_timestamp := VI_System_Time_MS;
          
END_FUNCTION_BLOCK

FUNCTION_BLOCK FB_Gas_Smoke_Manager
  VAR_INPUT
    VI_System_Time_MS : UDINT;
    VI_IsActivePLC : BOOL;
    VI_Mute_Request : BOOL;
  END_VAR
  VAR_OUTPUT
    VO_Smoke_Detected : BOOL;
    VO_Gas_Detected : BOOL;
    VO_CO_Warning_Level : BOOL;
    VO_CO_Alarm_Level : BOOL;
    VO_Status_Msg : STRING(200);
  END_VAR
  VAR_IN_OUT
    VI_Methane_LEL : ARRAY[1..GVL_CONSTANTS.C_MAX_METHANE_SENSORS] OF REAL;
    VI_CO_PPM : ARRAY[1..GVL_CONSTANTS.C_MAX_CO_SENSORS] OF REAL;
    VI_Smoke_Sensors : ARRAY[1..GVL_CONSTANTS.C_MAX_SMOKE_SENSORS] OF BOOL;
  END_VAR
  VAR
    L_Methane_Max : REAL;
    L_CO_Max : REAL;
    L_Smoke_Count : UINT;
    L_Smoke_Active : BOOL;
    L_i : INT;
    L_CO_Timer_30ppm : FB_System_Timer;
    L_CO_Timer_70ppm : FB_System_Timer;
    L_CO_Timer_400ppm : FB_System_Timer;
    L_CO_Level_30 : BOOL;
    L_CO_Level_70 : BOOL;
    L_CO_Level_400 : BOOL;
    L_Smoke_Timer : ARRAY[1..GVL_CONSTANTS.C_MAX_SMOKE_SENSORS] OF FB_System_Timer;
  END_VAR

            IF NOT VI_IsActivePLC THEN RETURN; END_IF;

// Reset outputs
VO_Smoke_Detected := FALSE;
VO_Gas_Detected := FALSE;
VO_CO_Warning_Level := FALSE;
VO_CO_Alarm_Level := FALSE;
VO_Status_Msg := 'ОК';

// --- Methane ---
L_Methane_Max := 0.0;
FOR L_i := 1 TO GVL_CONSTANTS.C_MAX_METHANE_SENSORS DO
    IF VI_Methane_LEL[L_i] > L_Methane_Max THEN
        L_Methane_Max := VI_Methane_LEL[L_i];
    END_IF;
END_FOR;

IF L_Methane_Max >= 20.0 THEN
    VO_Gas_Detected := TRUE;
END_IF;

// --- CO ---
L_CO_Max := 0.0;
FOR L_i := 1 TO GVL_CONSTANTS.C_MAX_CO_SENSORS DO
    IF VI_CO_PPM[L_i] > L_CO_Max THEN
        L_CO_Max := VI_CO_PPM[L_i];
    END_IF;
END_FOR;

L_CO_Level_30 := (L_CO_Max >= 30.0);
L_CO_Level_70 := (L_CO_Max >= 70.0);
L_CO_Level_400 := (L_CO_Max >= 400.0);

L_CO_Timer_30ppm(IN := L_CO_Level_30, PT := T#8h, VI_System_Time_MS := VI_System_Time_MS);
L_CO_Timer_70ppm(IN := L_CO_Level_70, PT := T#1h, VI_System_Time_MS := VI_System_Time_MS);
L_CO_Timer_400ppm(IN := L_CO_Level_400, PT := T#15m, VI_System_Time_MS := VI_System_Time_MS);

IF L_CO_Timer_30ppm.Q THEN
    VO_CO_Warning_Level := TRUE;
END_IF;

IF L_CO_Timer_70ppm.Q OR L_CO_Timer_400ppm.Q THEN
    VO_CO_Alarm_Level := TRUE;
END_IF;

// --- Smoke ---
L_Smoke_Count := 0;
L_Smoke_Active := FALSE;

FOR L_i := 1 TO GVL_CONSTANTS.C_MAX_SMOKE_SENSORS DO
    L_Smoke_Timer[L_i](IN := VI_Smoke_Sensors[L_i], PT := T#30s, VI_System_Time_MS := VI_System_Time_MS);

    IF VI_Smoke_Sensors[L_i] THEN
        L_Smoke_Count := L_Smoke_Count + 1;
    END_IF;

    IF L_Smoke_Timer[L_i].Q OR (L_Smoke_Count >= 2) THEN
        L_Smoke_Active := TRUE;
    END_IF;
END_FOR;

IF L_Smoke_Active THEN
    VO_Smoke_Detected := TRUE;
END_IF;

// Status
IF VO_Smoke_Detected THEN
    VO_Status_Msg := 'ПОЖАР';
ELSIF VO_Gas_Detected THEN
    VO_Status_Msg := 'УТЕЧКА ГАЗА';
ELSIF VO_CO_Alarm_Level THEN
    VO_Status_Msg := 'КРИТИЧЕСКИЙ CO';
ELSIF VO_CO_Warning_Level THEN
    VO_Status_Msg := 'ПОВЫШЕННЫЙ CO';
ELSE
    VO_Status_Msg := 'ОК';
END_IF;
// >>> BULK_SYNC_ANCHOR: FB_Gas_Smoke_Manager <<<
          
END_FUNCTION_BLOCK

FUNCTION_BLOCK FB_PID_Controller
  VAR_INPUT
    VI_SetPoint : REAL;
    VI_ProcessValue : REAL;
    VI_Kp : REAL;
    VI_Tn : REAL;
    VI_Tv : REAL;
    VI_Y_Min : REAL := 0.0;
    VI_Y_Max : REAL := 100.0;
    VI_Manual_Mode : BOOL;
    VI_Manual_Value : REAL;
    VI_Deadband : REAL := 0.1;
    VI_Cycle_Time_S : REAL := 0.01;
    VI_Reset : BOOL;
  END_VAR
  VAR_OUTPUT
    VO_Output : REAL;
    VO_Error : REAL;
    VO_Limiting : BOOL;
  END_VAR
  VAR
    L_Integral_Sum : REAL;
    L_Prev_Error : REAL;
    L_Derivative : REAL;
    L_Output_Raw : REAL;
  END_VAR

            // Расчет ошибки
VO_Error := VI_SetPoint - VI_ProcessValue;

// Проверка мертвой зоны
IF ABS(VO_Error) < VI_Deadband THEN
    VO_Error := 0.0;
END_IF;

IF VI_Reset THEN
    L_Integral_Sum := 0.0;
    L_Prev_Error := 0.0;
    VO_Output := 0.0;
    RETURN;
END_IF;

IF VI_Manual_Mode THEN
    VO_Output := VI_Manual_Value;
    // Безударный переход: при выходе из ручного режима выход должен остаться прежним.
    // Так как Выход = P + I + D, то I = Выход - P - D.
    // Для простоты D при переходе обнуляем (или игнорируем), тогда I = Выход - P.
    L_Integral_Sum := VO_Output - (VI_Kp * VO_Error);
    L_Prev_Error := VO_Error;
    RETURN;
END_IF;

// Пропорциональная составляющая
L_Output_Raw := VI_Kp * VO_Error;

// Интегральная составляющая (Метод трапеций)
IF VI_Tn > 0.0 THEN
    // Anti-windup: не накапливаем интеграл, если выход уже на пределе и ошибка того же знака
    IF NOT VO_Limiting OR (VO_Error > 0.0 AND L_Output_Raw < VI_Y_Max) OR (VO_Error < 0.0 AND L_Output_Raw > VI_Y_Min) THEN
        L_Integral_Sum := L_Integral_Sum + (VI_Kp / VI_Tn) * VO_Error * VI_Cycle_Time_S;
    END_IF;
    L_Output_Raw := L_Output_Raw + L_Integral_Sum;
END_IF;

// Дифференциальная составляющая
IF VI_Tv > 0.0 THEN
    L_Derivative := (VO_Error - L_Prev_Error) / VI_Cycle_Time_S;
    L_Output_Raw := L_Output_Raw + VI_Kp * VI_Tv * L_Derivative;
END_IF;

L_Prev_Error := VO_Error;

// Ограничение выхода
IF L_Output_Raw > VI_Y_Max THEN
    VO_Output := VI_Y_Max;
    VO_Limiting := TRUE;
ELSIF L_Output_Raw < VI_Y_Min THEN
    VO_Output := VI_Y_Min;
    VO_Limiting := TRUE;
ELSE
    VO_Output := L_Output_Raw;
    VO_Limiting := FALSE;
END_IF;
// >>> BULK_SYNC_ANCHOR: FB_PID_Controller <<<
          
END_FUNCTION_BLOCK

FUNCTION_BLOCK FB_Gateway_Interface
  VAR_INPUT
    VI_System_Time_MS : UDINT;
    VI_Local_PLC_Role : E_PLC_ROLE;
    VI_Incoming_Command : ST_Gateway_Command;
    VI_Command_Received : BOOL;
    VI_Outdoor_Temp : REAL;
    VI_Security_Armed : BOOL;
    VI_Flood_Alarm_Active : BOOL;
    VI_Gas_Alarm_Active : BOOL;
    VI_Fire_Alarm_Active : BOOL;
    VI_Methane_Concentration : REAL;
    VI_Active_Scenario : E_SCENARIO_TYPE;
    VI_Send_2FA_Req : BOOL;
    VI_2FA_Code : STRING(6);
  END_VAR
  VAR_OUTPUT
    VO_Modbus_Registers : ARRAY[0..GVL_CONSTANTS.C_MAX_MODBUS_REGISTERS-1] OF WORD;
    VO_Lighting_Override : ARRAY[1..32] OF BYTE;
    VO_Blinds_Override : ARRAY[1..GVL_CONSTANTS.C_MAX_BLINDS] OF BYTE;
    VO_Socket_Override : ARRAY[1..GVL_CONSTANTS.C_MAX_SOCKETS] OF BOOL;
    VO_Arm_Req : BOOL;
    VO_Disarm_Req : BOOL;
    VO_PIN_Code : STRING(4);
    VO_RFID_Tag : STRING(20);
    VO_2FA_Code_In : STRING(6);
    VO_Data_Ready : BOOL;
    VO_HMI_Status_Message : STRING(200);
    VO_Telegram_Msg : STRING(200);
    VO_Send_Telegram : BOOL;
    VO_Set_Scenario_Req : BOOL;
    VO_Target_Scenario : E_SCENARIO_TYPE;
    VO_Set_Temp_Req : BOOL;
    VO_Target_Zone : INT;
    VO_Target_Temp : REAL;
    VO_Set_Vent_Req : BOOL;
    VO_Target_Vent_Speed : BYTE;
    VO_Reset_Errors_Req : BOOL;
    VO_Set_Config_Req : BOOL;
    VO_Sync_Time_Req : BOOL;
    VO_New_Time_MS : UDINT;
  END_VAR
  VAR_IN_OUT
    VI_FloorHeating_Temps : ARRAY[1..8] OF REAL;
    VI_Room_Temps : ARRAY[1..16] OF REAL;
    VI_Zone_Valve_States : ARRAY[1..8] OF BOOL;
    VI_Manifold_Pressures : ARRAY[1..GVL_CONSTANTS.C_MAX_MANIFOLDS] OF REAL;
    VI_Manifold_Pump_States : ARRAY[1..GVL_CONSTANTS.C_MAX_MANIFOLDS] OF BOOL;
    VI_Lighting_Base_Levels : ARRAY[1..32] OF BYTE;
    VI_Socket_States : ARRAY[1..GVL_CONSTANTS.C_MAX_SOCKETS] OF BOOL;
    VI_Blinds_Positions : ARRAY[1..GVL_CONSTANTS.C_MAX_BLINDS] OF BYTE;
    VI_Allowed_IPs : ARRAY[1..GVL_CONSTANTS.C_MAX_ALLOWED_IPS] OF STRING(15);
  END_VAR
  VAR
    L_last_update_time : UDINT;
    L_i : INT;
    L_j : INT;
    L_idx : INT;
    L_tmp_word : WORD;
    L_Code_UDINT : UDINT;
    L_Prev_Fire : BOOL;
    L_Prev_Gas : BOOL;
    L_Prev_Flood : BOOL;
    L_Prev_Security : BOOL;
    L_Deduplicator : FB_Command_Deduplication;
    L_CRC_Calc : FB_CRC32_Calculator;
    L_Calculated_CRC : DWORD;
    L_Command_Size : UDINT;
    L_IP_Allowed : BOOL;
    L_Process_Command : ST_Gateway_Command;
    L_Has_Command_To_Process : BOOL;
  END_VAR
  VAR RETAIN
    L_Command_Buffer : ARRAY[1..GVL_CONSTANTS.C_MAX_GATEWAY_COMMANDS] OF ST_Gateway_Command;
    L_Buffer_Head : INT := 1;
    L_Buffer_Tail : INT := 1;
    L_Buffer_Count : INT := 0;
  END_VAR

            // Отправка уведомлений в Telegram (ТЗ 10.2)
VO_Send_Telegram := FALSE;
IF VI_Fire_Alarm_Active AND NOT L_Prev_Fire THEN
    VO_Telegram_Msg := 'ВНИМАНИЕ! ПОЖАРНАЯ ТРЕВОГА!';
    VO_Send_Telegram := TRUE;
END_IF;
IF VI_Gas_Alarm_Active AND NOT L_Prev_Gas THEN
    VO_Telegram_Msg := 'ВНИМАНИЕ! УТЕЧКА ГАЗА!';
    VO_Send_Telegram := TRUE;
END_IF;
IF VI_Flood_Alarm_Active AND NOT L_Prev_Flood THEN
    VO_Telegram_Msg := 'ВНИМАНИЕ! ПРОТЕЧКА ВОДЫ!';
    VO_Send_Telegram := TRUE;
END_IF;
IF VI_Security_Armed AND NOT L_Prev_Security THEN
    VO_Telegram_Msg := 'ОХРАНА ВКЛЮЧЕНА';
    VO_Send_Telegram := TRUE;
ELSIF NOT VI_Security_Armed AND L_Prev_Security THEN
    VO_Telegram_Msg := 'ОХРАНА ОТКЛЮЧЕНА';
    VO_Send_Telegram := TRUE;
END_IF;

L_Prev_Fire := VI_Fire_Alarm_Active;
L_Prev_Gas := VI_Gas_Alarm_Active;
L_Prev_Flood := VI_Flood_Alarm_Active;
L_Prev_Security := VI_Security_Armed;

// Обновление данных Modbus (раз в 1 сек)
IF (VI_System_Time_MS - L_last_update_time) >= GVL_CONSTANTS.C_MS_IN_SECOND THEN
    L_last_update_time := VI_System_Time_MS;
    
    // 0: Статус ПЛК и Аварии
    L_tmp_word := 0;
    IF VI_Local_PLC_Role = E_PLC_ROLE.ROLE_ACTIVE THEN L_tmp_word := L_tmp_word OR 1; END_IF;
    IF VI_Security_Armed THEN L_tmp_word := L_tmp_word OR 2; END_IF;
    IF VI_Flood_Alarm_Active THEN L_tmp_word := L_tmp_word OR 4; END_IF;
    IF VI_Gas_Alarm_Active THEN L_tmp_word := L_tmp_word OR 8; END_IF;
    IF VI_Fire_Alarm_Active THEN L_tmp_word := L_tmp_word OR 16; END_IF;
    VO_Modbus_Registers[0] := L_tmp_word;

    // 1-16: Температуры пола (x10)
    FOR L_i := 1 TO 8 DO
        VO_Modbus_Registers[L_i] := TO_WORD(TO_INT(VI_FloorHeating_Temps[L_i] * 10.0));
    END_FOR;

    // 17-310102: Температуры помещений (x10)
    FOR L_i := 1 TO 16 DO
        VO_Modbus_Registers[16 + L_i] := TO_WORD(TO_INT(VI_Room_Temps[L_i] * 10.0));
    END_FOR;

    // 310103: Состояние клапанов зон (битовая маска 1-16)
    L_tmp_word := 0;
    FOR L_i := 1 TO 8 DO
        IF VI_Zone_Valve_States[L_i] THEN
            L_tmp_word := L_tmp_word OR SHL(TO_WORD(1), L_i - 1);
        END_IF;
    END_FOR;
    VO_Modbus_Registers[33] := L_tmp_word;

    // 34-38: Давление в коллекторах (x100)
    FOR L_i := 1 TO GVL_CONSTANTS.C_MAX_MANIFOLDS DO
        VO_Modbus_Registers[33 + L_i] := TO_WORD(TO_INT(VI_Manifold_Pressures[L_i] * 100.0));
    END_FOR;

    // 40-55: Базовое освещение
    FOR L_i := 1 TO 32 DO
        VO_Modbus_Registers[39 + L_i] := TO_WORD(VI_Lighting_Base_Levels[L_i]);
    END_FOR;

    // 60-79: Положение штор (20 шт)
    FOR L_i := 1 TO GVL_CONSTANTS.C_MAX_BLINDS DO
        VO_Modbus_Registers[59 + L_i] := TO_WORD(VI_Blinds_Positions[L_i]);
    END_FOR;

    // 80-82: Розетки (битовая маска, 36 розеток -> 3 WORD)
    FOR L_i := 0 TO (GVL_CONSTANTS.C_MAX_SOCKETS - 1) / 16 DO
        L_tmp_word := 0;
        FOR L_j := 1 TO 16 DO
            L_idx := (L_i * 16) + L_j;
            IF L_idx <= GVL_CONSTANTS.C_MAX_SOCKETS THEN
                IF VI_Socket_States[L_idx] THEN
                    L_tmp_word := L_tmp_word OR SHL(TO_WORD(1), L_j - 1);
                END_IF;
            END_IF;
        END_FOR;
        VO_Modbus_Registers[79 + L_i] := L_tmp_word;
    END_FOR;

    // 100-102: 2FA Request and Code
    VO_Modbus_Registers[100] := SEL(VI_Send_2FA_Req, 0, 1);
    IF VI_Send_2FA_Req THEN
        L_Code_UDINT := STRING_TO_UDINT(VI_2FA_Code);
        VO_Modbus_Registers[101] := TO_WORD(L_Code_UDINT AND 16#FFFF);
        VO_Modbus_Registers[102] := TO_WORD(SHR(L_Code_UDINT, 16));
    ELSE
        VO_Modbus_Registers[101] := 0;
        VO_Modbus_Registers[102] := 0;
    END_IF;

    VO_Data_Ready := TRUE;
END_IF;

// Обработка входящих команд
VO_Arm_Req := FALSE;
VO_Disarm_Req := FALSE;
VO_Set_Scenario_Req := FALSE;
VO_Set_Temp_Req := FALSE;
VO_Set_Vent_Req := FALSE;
VO_Reset_Errors_Req := FALSE;
VO_Set_Config_Req := FALSE;
VO_Sync_Time_Req := FALSE;
L_Has_Command_To_Process := FALSE;

// 1. Прием команды и буферизация
IF VI_Command_Received THEN
    IF VI_Local_PLC_Role = E_PLC_ROLE.ROLE_ACTIVE THEN
        // Если активен, обрабатываем сразу
        L_Process_Command := VI_Incoming_Command;
        L_Has_Command_To_Process := TRUE;
    ELSE
        // Если резервный, добавляем в буфер
        IF L_Buffer_Count < GVL_CONSTANTS.C_MAX_GATEWAY_COMMANDS THEN
            L_Command_Buffer[L_Buffer_Head] := VI_Incoming_Command;
            L_Buffer_Head := L_Buffer_Head + 1;
            IF L_Buffer_Head > GVL_CONSTANTS.C_MAX_GATEWAY_COMMANDS THEN L_Buffer_Head := 1; END_IF;
            L_Buffer_Count := L_Buffer_Count + 1;
        END_IF;
    END_IF;
END_IF;

// 2. Извлечение из буфера при переходе в активный режим
IF NOT L_Has_Command_To_Process AND (VI_Local_PLC_Role = E_PLC_ROLE.ROLE_ACTIVE) AND (L_Buffer_Count > 0) THEN
    L_Process_Command := L_Command_Buffer[L_Buffer_Tail];
    L_Buffer_Tail := L_Buffer_Tail + 1;
    IF L_Buffer_Tail > GVL_CONSTANTS.C_MAX_GATEWAY_COMMANDS THEN L_Buffer_Tail := 1; END_IF;
    L_Buffer_Count := L_Buffer_Count - 1;
    L_Has_Command_To_Process := TRUE;
END_IF;

// 3. Обработка команды
IF L_Has_Command_To_Process THEN
    // Проверка IP-адреса источника
    L_IP_Allowed := FALSE;
    IF L_Process_Command.source_ip = '' THEN
        L_IP_Allowed := TRUE; // Если IP не передан, пропускаем (для обратной совместимости или локальных вызовов)
    ELSE
        FOR L_i := 1 TO GVL_CONSTANTS.C_MAX_ALLOWED_IPS DO
            IF VI_Allowed_IPs[L_i] = L_Process_Command.source_ip THEN
                L_IP_Allowed := TRUE;
                EXIT;
            END_IF;
        END_FOR;
    END_IF;
    
    IF NOT L_IP_Allowed THEN
        VO_HMI_Status_Message := 'Gateway: Ошибка безопасности (Неизвестный IP)';
        RETURN;
    END_IF;

    // Проверка целостности данных (CRC32)
    // Размер данных для расчета CRC: размер структуры минус размер самого поля crc32
    L_Command_Size := SIZEOF(L_Process_Command) - SIZEOF(L_Process_Command.crc32);
    L_Calculated_CRC := L_CRC_Calc.Calculate();
    
    IF L_Calculated_CRC = L_Process_Command.crc32 THEN
        L_Deduplicator(
            VI_Command_ID := L_Process_Command.command_id,
            VI_Command_Type := L_Process_Command.command_type,
            VI_Command_Value := L_Process_Command.target_value,
            VI_System_Time_MS := VI_System_Time_MS
        );
        
        IF L_Deduplicator.VO_Is_New_Command THEN
            CASE L_Process_Command.command_type OF
        E_Gateway_Command_Type.CMD_SET_SCENARIO: // Управление сценариями
            VO_Set_Scenario_Req := TRUE;
            VO_Target_Scenario := L_Process_Command.target_scenario;
            VO_HMI_Status_Message := 'Gateway: Сценарий изменен';
        E_Gateway_Command_Type.CMD_SET_LIGHT: // Управление освещением
            IF (L_Process_Command.target_zone >= 1) AND (L_Process_Command.target_zone <= 32) THEN
                VO_Lighting_Override[L_Process_Command.target_zone] := TO_BYTE(L_Process_Command.target_value);
                VO_HMI_Status_Message := 'Gateway: Команда освещения принята';
            END_IF;
        E_Gateway_Command_Type.CMD_SET_BLINDS: // Управление шторами
            IF (L_Process_Command.target_zone >= 1) AND (L_Process_Command.target_zone <= GVL_CONSTANTS.C_MAX_BLINDS) THEN
                VO_Blinds_Override[L_Process_Command.target_zone] := TO_BYTE(L_Process_Command.target_value);
                VO_HMI_Status_Message := 'Gateway: Команда штор принята';
            END_IF;
        E_Gateway_Command_Type.CMD_SET_SOCKET: // Розетки
            IF (L_Process_Command.target_zone >= 1) AND (L_Process_Command.target_zone <= GVL_CONSTANTS.C_MAX_SOCKETS) THEN
                VO_Socket_Override[L_Process_Command.target_zone] := L_Process_Command.target_on_off;
                VO_HMI_Status_Message := 'Gateway: Команда розетки принята';
            END_IF;
        E_Gateway_Command_Type.CMD_SET_SECURITY: // Охрана
            IF L_Process_Command.target_armed THEN
                VO_Arm_Req := TRUE;
            ELSE
                VO_Disarm_Req := TRUE;
            END_IF;
            VO_PIN_Code := L_Process_Command.target_pin;
            VO_2FA_Code_In := L_Process_Command.target_2fa_code;
            VO_HMI_Status_Message := 'Gateway: Запрос охраны принят';
        E_Gateway_Command_Type.CMD_SET_TEMP: // Управление температурой
            IF (L_Process_Command.target_zone >= 1) AND (L_Process_Command.target_zone <= 32) THEN
                VO_Set_Temp_Req := TRUE;
                VO_Target_Zone := L_Process_Command.target_zone;
                VO_Target_Temp := L_Process_Command.target_value;
                VO_HMI_Status_Message := 'Gateway: Уставка температуры изменена';
            END_IF;
        E_Gateway_Command_Type.CMD_SET_VENT: // Управление вентиляцией
            // Пример: изменение скорости притока
            VO_Set_Vent_Req := TRUE;
            VO_Target_Vent_Speed := TO_BYTE(L_Process_Command.target_value);
            VO_HMI_Status_Message := 'Gateway: Уставка вентиляции изменена';
        E_Gateway_Command_Type.CMD_TELEGRAM_MSG: // Отправка сообщения в Telegram
            VO_Telegram_Msg := L_Process_Command.telegram_msg;
            VO_Send_Telegram := TRUE;
            VO_HMI_Status_Message := 'Gateway: Сообщение Telegram отправлено';

        E_Gateway_Command_Type.CMD_SYNC_TIME: // Синхронизация времени
            VO_Sync_Time_Req := TRUE;
            VO_New_Time_MS := TO_UDINT(L_Process_Command.target_value);
            VO_HMI_Status_Message := 'Gateway: Время синхронизировано';

        E_Gateway_Command_Type.CMD_RESET_ERRORS: // Квитирование / сброс ошибок
            VO_Reset_Errors_Req := TRUE;
            VO_HMI_Status_Message := 'Gateway: Запрос на сброс ошибок принят';

        E_Gateway_Command_Type.CMD_SET_CONFIG: // Применение конфигурации
            VO_Set_Config_Req := TRUE;
            VO_HMI_Status_Message := 'Gateway: Запрос на применение конфигурации принят';
        END_CASE;
    END_IF;
ELSE
    VO_HMI_Status_Message := 'Gateway: Ошибка CRC команды';
END_IF;
END_IF;
// >>> BULK_SYNC_ANCHOR: FB_Gateway_Interface <<<
          
END_FUNCTION_BLOCK

FUNCTION_BLOCK FB_Valve_Test_Manager
  VAR_INPUT
    VI_System_Time_MS : UDINT;
    VI_IsActivePLC : BOOL;
  END_VAR
  VAR_OUTPUT
    VO_Test_Active : BOOL;
    VO_Current_Valve : INT;
    VO_Valve_Cmd : ARRAY[1..GVL_CONSTANTS.C_MAX_MANIFOLDS] OF BOOL;
    VO_Test_Results : ARRAY[1..GVL_CONSTANTS.C_MAX_MANIFOLDS] OF BOOL;
    VO_Status_Msg : STRING(200);
  END_VAR
  VAR_IN_OUT
    VI_Valve_Currents : ARRAY[1..GVL_CONSTANTS.C_MAX_MANIFOLDS] OF REAL;
    VI_Valve_End_Switches : ARRAY[1..GVL_CONSTANTS.C_MAX_MANIFOLDS] OF BOOL;
    VI_Config : ARRAY[1..GVL_CONSTANTS.C_MAX_MANIFOLDS] OF ST_Valve_Test_Config;
  END_VAR
  VAR
    L_State : INT;
    L_Current_Valve : INT := 1;
    L_Test_Start_Time : UDINT;
    L_Last_Test_Time : ARRAY[1..GVL_CONSTANTS.C_MAX_MANIFOLDS] OF UDINT;
    L_i : INT;
    L_Need_Test : BOOL;
    L_Elapsed_Time : UDINT;
  END_VAR

            IF NOT VI_IsActivePLC THEN RETURN; END_IF;

CASE L_State OF
    0: // Ожидание
        VO_Test_Active := FALSE;
        L_Need_Test := FALSE;
        
        // Поиск клапана, которому нужен тест (раз в неделю)
        FOR L_i := 1 TO GVL_CONSTANTS.C_MAX_MANIFOLDS DO
            IF VI_Config[L_i].enabled AND ((VI_System_Time_MS - L_Last_Test_Time[L_i]) > (VI_Config[L_i].test_interval_days * 86400000)) THEN
                L_Current_Valve := L_i;
                L_Need_Test := TRUE;
                EXIT;
            END_IF;
        END_FOR;
        
        IF L_Need_Test THEN
            L_State := 1;
            L_Test_Start_Time := VI_System_Time_MS;
            VO_Test_Active := TRUE;
            VO_Current_Valve := L_Current_Valve;
            VO_Valve_Cmd[L_Current_Valve] := TRUE; // Открываем
            VO_Status_Msg := CONCAT('ТЕСТ КЛАПАНА ', INT_TO_STRING(L_Current_Valve));
            VO_Test_Results[L_Current_Valve] := TRUE; // Сброс результата
        END_IF;
        
    1: // Тестирование (ожидание открытия)
        L_Elapsed_Time := (VI_System_Time_MS - L_Test_Start_Time);
        
        IF VI_Valve_End_Switches[L_Current_Valve] THEN
            // Концевик сработал до истечения таймаута
            // Проверка тока
            IF ABS(VI_Valve_Currents[L_Current_Valve] - VI_Config[L_Current_Valve].Nominal_Current) > (VI_Config[L_Current_Valve].Nominal_Current * 0.2) THEN
                VO_Test_Results[L_Current_Valve] := FALSE; // Ошибка по току
            END_IF;
            
            GVL_Retain.G_Valve_Test_Results[L_Current_Valve] := VO_Test_Results[L_Current_Valve];
            
            VO_Valve_Cmd[L_Current_Valve] := FALSE; // Закрываем
            L_Test_Start_Time := VI_System_Time_MS; // Перезапускаем таймер для проверки закрытия
            L_State := 2;
        ELSIF L_Elapsed_Time > TO_UDINT(VI_Config[L_Current_Valve].nominal_close_time_sec * 1000.0) THEN
            // Таймаут открытия (заклинивание)
            VO_Test_Results[L_Current_Valve] := FALSE; 
            GVL_Retain.G_Valve_Test_Results[L_Current_Valve] := FALSE;
            VO_Status_Msg := CONCAT('ОШИБКА: ЗАКЛИНИВАНИЕ КЛАПАНА ', INT_TO_STRING(L_Current_Valve));
            
            VO_Valve_Cmd[L_Current_Valve] := FALSE; // Закрываем
            L_Test_Start_Time := VI_System_Time_MS; // Перезапускаем таймер
            L_State := 2;
        END_IF;
        
    2: // Ожидание закрытия
        L_Elapsed_Time := (VI_System_Time_MS - L_Test_Start_Time);
        
        IF NOT VI_Valve_End_Switches[L_Current_Valve] THEN
            // Концевик разомкнулся (клапан закрыт)
            L_Last_Test_Time[L_Current_Valve] := VI_System_Time_MS;
            L_State := 0;
            IF VO_Test_Results[L_Current_Valve] THEN
                VO_Status_Msg := 'ТЕСТ ЗАВЕРШЕН УСПЕШНО';
            END_IF;
        ELSIF L_Elapsed_Time > TO_UDINT(VI_Config[L_Current_Valve].nominal_close_time_sec * 1000.0) THEN
            // Таймаут закрытия (заклинивание)
            VO_Test_Results[L_Current_Valve] := FALSE; 
            GVL_Retain.G_Valve_Test_Results[L_Current_Valve] := FALSE;
            VO_Status_Msg := CONCAT('ОШИБКА: НЕ ЗАКРЫЛСЯ КЛАПАН ', INT_TO_STRING(L_Current_Valve));
            
            L_Last_Test_Time[L_Current_Valve] := VI_System_Time_MS;
            L_State := 0;
        END_IF;
END_CASE;
          
END_FUNCTION_BLOCK

FUNCTION_BLOCK FB_System_Intent_Publisher
  VAR_INPUT
    VI_System_Time_MS : UDINT;
    VI_Gateway_Writes_Allowed : BOOL;
  END_VAR

            // ==============================================================================
// System intent publisher helper
//
// Internal helper for PRG_System.
// Owns publication of system-mode gates into GVL_INTENT_SYSTEM.
// ==============================================================================



GVL_INTENT_SYSTEM.I_Source_Valid := TRUE;
GVL_INTENT_SYSTEM.I_Last_Update_MS := VI_System_Time_MS;
GVL_INTENT_SYSTEM.I_Mode_Safe_Stop_Active := (GVL_STATE.G_System_Mode = E_System_Operating_Mode.MODE_SAFE_STOP);
GVL_INTENT_SYSTEM.I_Mode_Degraded_Active := (GVL_STATE.G_System_Mode = E_System_Operating_Mode.MODE_DEGRADED);
GVL_INTENT_SYSTEM.I_Mode_Freeze_Protection_Active := (GVL_STATE.G_System_Mode = E_System_Operating_Mode.MODE_FREEZE_PROTECTION);
GVL_INTENT_SYSTEM.I_Operator_Scenario_Block := (GVL_STATE.G_System_Mode = E_System_Operating_Mode.MODE_SAFE_STOP);
GVL_INTENT_SYSTEM.I_Lighting_Overrides_Block := (GVL_STATE.G_System_Mode = E_System_Operating_Mode.MODE_SAFE_STOP);
GVL_INTENT_SYSTEM.I_Blinds_Overrides_Block := (GVL_STATE.G_System_Mode = E_System_Operating_Mode.MODE_SAFE_STOP);
GVL_INTENT_SYSTEM.I_Socket_Overrides_Block := (GVL_STATE.G_System_Mode = E_System_Operating_Mode.MODE_SAFE_STOP);
GVL_INTENT_SYSTEM.I_Gateway_Writes_Allowed := VI_Gateway_Writes_Allowed;
GVL_INTENT_SYSTEM.I_Scenario_Request_Allowed := (GVL_STATE.G_System_Mode <> E_System_Operating_Mode.MODE_SAFE_STOP);

// >>> BULK_SYNC_ANCHOR: FB_System_Intent_Publisher <<<
          
END_FUNCTION_BLOCK

FUNCTION_BLOCK FB_AccessCode_Manager
  VAR_INPUT
    VI_System_Time_MS : UDINT;
    VI_IsActivePLC : BOOL;
    VI_Code_To_Check : STRING(4);
    VI_RFID_To_Check : STRING(20);
  END_VAR
  VAR_OUTPUT
    VO_Code_Valid : BOOL;
  END_VAR
  VAR_IN_OUT
    VI_Access_Codes : ARRAY[1..GVL_CONSTANTS.C_MAX_ACCESS_CODES] OF DWORD;
    VI_RFID_Tags : ARRAY[1..GVL_CONSTANTS.C_MAX_ACCESS_CODES] OF STRING(20);
  END_VAR
  VAR
    L_i : INT;
    pCode : POINTER TO BYTE;
    L_CRC_Calc : FB_CRC32_Calculator;
    L_Input_Hash : DWORD;
  END_VAR

            VO_Code_Valid := FALSE;

// Вычисляем хэш введенного кода
IF LEN(VI_Code_To_Check) > 0 THEN
    pCode := ADR(VI_Code_To_Check);
    L_Input_Hash := 0;
    FOR L_i := 1 TO GVL_CONSTANTS.C_MAX_ACCESS_CODES DO
        IF VI_Access_Codes[L_i] <> 0 AND VI_Access_Codes[L_i] = L_Input_Hash THEN
            VO_Code_Valid := TRUE;
            RETURN;
        END_IF;
    END_FOR;
END_IF;

// Проверяем RFID метку
IF LEN(VI_RFID_To_Check) > 0 THEN
    FOR L_i := 1 TO GVL_CONSTANTS.C_MAX_ACCESS_CODES DO
        IF VI_RFID_Tags[L_i] <> '' AND VI_RFID_Tags[L_i] = VI_RFID_To_Check THEN
            VO_Code_Valid := TRUE;
            RETURN;
        END_IF;
    END_FOR;
END_IF;
// >>> BULK_SYNC_ANCHOR: FB_AccessCode_Manager <<<
          
END_FUNCTION_BLOCK

FUNCTION_BLOCK FB_Device_Predictive_Diag
  VAR_INPUT
    VI_Current_Value : REAL;
    VI_Nominal_Value : REAL;
    VI_Is_Running : BOOL;
    VI_Reset_Stats : BOOL;
    VI_System_Time_MS : UDINT;
  END_VAR
  VAR_IN_OUT
    VIO_Health_Data : ST_Device_Health;
  END_VAR
  VAR
    L_Prev_Running : BOOL;
    L_Start_Time : UDINT;
    L_Last_Calc_Time : UDINT;
    L_Elapsed_MS : UDINT;
    L_Accumulated_MS : UDINT;
    L_Timer_Running : FB_System_Timer;
  END_VAR

            // 0. Сброс статистики
IF VI_Reset_Stats THEN
    VIO_Health_Data.Starts_Count := 0;
    VIO_Health_Data.Sample_Count := 0;
    VIO_Health_Data.Current_Sum := 0.0;
    VIO_Health_Data.Avg_Start_Current := 0.0;
    VIO_Health_Data.Health_Score := 100;
    VIO_Health_Data.Maintenance_Required := FALSE;
    VIO_Health_Data.Warning_Message := '';
    VIO_Health_Data.Last_Start_Current := 0.0;
    VIO_Health_Data.Total_Runtime_Hours := 0;
    L_Accumulated_MS := 0;
END_IF;

// 1. Счётчик пусков и замер пускового тока
IF VI_Is_Running AND NOT L_Prev_Running THEN
    VIO_Health_Data.Starts_Count := VIO_Health_Data.Starts_Count + 1;
    VIO_Health_Data.Last_Start_Current := VI_Current_Value;
    L_Start_Time := VI_System_Time_MS;
    L_Last_Calc_Time := VI_System_Time_MS;
    
    // Обновление среднего пускового тока
    VIO_Health_Data.Sample_Count := VIO_Health_Data.Sample_Count + 1;
    VIO_Health_Data.Current_Sum := VIO_Health_Data.Current_Sum + VI_Current_Value;
    VIO_Health_Data.Avg_Start_Current := VIO_Health_Data.Current_Sum / UDINT_TO_REAL(VIO_Health_Data.Sample_Count);
    
    // 2. Анализ отклонения пускового тока (п. 12.1 ТЗ)
    IF VI_Current_Value > (VI_Nominal_Value * 1.5) THEN
        VIO_Health_Data.Health_Score := TO_BYTE(LIMIT(0, TO_INT(VIO_Health_Data.Health_Score) - 5, 100));
    ELSIF VI_Current_Value > (VI_Nominal_Value * 1.2) THEN
        VIO_Health_Data.Health_Score := TO_BYTE(LIMIT(0, TO_INT(VIO_Health_Data.Health_Score) - 1, 100));
    ELSIF VI_Current_Value < (VI_Nominal_Value * 0.5) THEN
        VIO_Health_Data.Health_Score := TO_BYTE(LIMIT(0, TO_INT(VIO_Health_Data.Health_Score) - 2, 100));
    END_IF;
END_IF;

// 3. Анализ рабочего тока и наработки
IF VI_Is_Running THEN
    L_Elapsed_MS := (VI_System_Time_MS - L_Last_Calc_Time);
    L_Accumulated_MS := L_Accumulated_MS + L_Elapsed_MS;
    L_Last_Calc_Time := VI_System_Time_MS;
    
    // Обновляем наработку каждый час (3600000 мс)
    IF L_Accumulated_MS >= 3600000 THEN
        VIO_Health_Data.Total_Runtime_Hours := VIO_Health_Data.Total_Runtime_Hours + 1;
        L_Accumulated_MS := L_Accumulated_MS - 3600000;
        
        // Естественный износ: -1% здоровья каждые 1000 часов
        IF (VIO_Health_Data.Total_Runtime_Hours MOD 1000) = 0 THEN
            VIO_Health_Data.Health_Score := TO_BYTE(LIMIT(0, TO_INT(VIO_Health_Data.Health_Score) - 1, 100));
        END_IF;
        
        // Анализ рабочего тока (после пускового режима)
        IF (VI_System_Time_MS - L_Start_Time) > 10000 THEN // 10 секунд после пуска
            IF VI_Current_Value > (VI_Nominal_Value * 1.1) THEN
                // Повышенный рабочий ток - ускоренный износ (-1% в час)
                VIO_Health_Data.Health_Score := TO_BYTE(LIMIT(0, TO_INT(VIO_Health_Data.Health_Score) - 1, 100));
            END_IF;
        END_IF;
    END_IF;
END_IF;

// 4. Генерация предупреждения
IF VIO_Health_Data.Health_Score < 20 THEN
    VIO_Health_Data.Maintenance_Required := TRUE;
    VIO_Health_Data.Warning_Message := 'Критический износ: проверьте механику';
ELSIF VIO_Health_Data.Health_Score < 60 THEN
    VIO_Health_Data.Maintenance_Required := FALSE;
    VIO_Health_Data.Warning_Message := 'Предупреждение: повышенное трение';
ELSE
    VIO_Health_Data.Maintenance_Required := FALSE;
    VIO_Health_Data.Warning_Message := 'В норме';
END_IF;

L_Prev_Running := VI_Is_Running;
          
END_FUNCTION_BLOCK

FUNCTION_BLOCK FB_System_Scenario_Arbitration
  VAR_INPUT
    VI_System_Time_MS : UDINT;
    VI_IsActivePLC : BOOL;
    VI_System_Mode : E_System_Operating_Mode;
    VI_Security_Armed : BOOL;
  END_VAR
  VAR_IN_OUT
    VIO_Scenario_Req_Operator : E_SCENARIO_TYPE;
    VIO_Scenario_Req_Gateway : E_SCENARIO_TYPE;
    VIO_Scenario_Req_Rule : E_SCENARIO_TYPE;
    VIO_Scenario_Req_Final : E_SCENARIO_TYPE;
    VIO_Scenario_Intent : E_SCENARIO_TYPE;
    VIO_Scenario_Source : E_SCENARIO_SOURCE;
  END_VAR
  VAR
    fbLogEvent : FB_LogEvent;
    fbScenarioManager : FB_Scenario_Manager;
  END_VAR

            // ==============================================================================
// System scenario arbitration helper
//
// Internal helper for PRG_System.
// Owns scenario request validation, priority resolution, fail-safe clamp,
// degraded-mode adaptation, policy logging, and FB_Scenario_Manager call.
// ==============================================================================



// === SCENARIO REQUEST VALIDATION ===
// Normalize invalid values to NONE to avoid corrupt inputs.
// Actual enum range in E_SCENARIO_TYPE is 0..7.
IF TO_USINT(VIO_Scenario_Req_Operator) > 7 THEN
    VIO_Scenario_Req_Operator := E_SCENARIO_TYPE.SCENARIO_NONE;
END_IF;

IF TO_USINT(VIO_Scenario_Req_Gateway) > 7 THEN
    VIO_Scenario_Req_Gateway := E_SCENARIO_TYPE.SCENARIO_NONE;
END_IF;

IF TO_USINT(VIO_Scenario_Req_Rule) > 7 THEN
    VIO_Scenario_Req_Rule := E_SCENARIO_TYPE.SCENARIO_NONE;
END_IF;

// === SCENARIO PRIORITY RESOLUTION ===
// Produces VIO_Scenario_Req_Final (TRACE ONLY, not executed directly)
IF VI_System_Mode = E_System_Operating_Mode.MODE_SAFE_STOP THEN
    VIO_Scenario_Req_Final := 0;
    VIO_Scenario_Source := SRC_SAFETY;
ELSIF VIO_Scenario_Req_Operator <> 0 THEN
    VIO_Scenario_Req_Final := VIO_Scenario_Req_Operator;
    VIO_Scenario_Source := SRC_OPERATOR;
ELSIF VIO_Scenario_Req_Gateway <> 0 THEN
    VIO_Scenario_Req_Final := VIO_Scenario_Req_Gateway;
    VIO_Scenario_Source := SRC_GATEWAY;
ELSIF VIO_Scenario_Req_Rule <> 0 THEN
    VIO_Scenario_Req_Final := VIO_Scenario_Req_Rule;
    VIO_Scenario_Source := SRC_RULE;
ELSE
    VIO_Scenario_Req_Final := GVL_STATUS.G_Current_Scenario;
    VIO_Scenario_Source := SRC_NONE;
END_IF;

VIO_Scenario_Intent := VIO_Scenario_Req_Final;

// === FAIL-SAFE SCENARIO CLAMP ===
CASE VI_System_Mode OF
    E_System_Operating_Mode.MODE_SAFE_STOP:
        VIO_Scenario_Intent := E_SCENARIO_TYPE.SCENARIO_NONE;

    E_System_Operating_Mode.MODE_FREEZE_PROTECTION:
        VIO_Scenario_Intent := E_SCENARIO_TYPE.SCENARIO_NONE;

    E_System_Operating_Mode.MODE_DEGRADED:
        CASE VIO_Scenario_Intent OF
            E_SCENARIO_TYPE.SCENARIO_NONE,
            E_SCENARIO_TYPE.SCENARIO_PRESENCE,
            E_SCENARIO_TYPE.SCENARIO_AWAY,
            E_SCENARIO_TYPE.SCENARIO_SLEEP:
                ; // allowed in degraded
        ELSE
            VIO_Scenario_Intent := E_SCENARIO_TYPE.SCENARIO_NONE;
        END_CASE;
END_CASE;

// === CONTEXT FAIL-SAFE AUTOMATION ===
// If security is armed and no explicit source is requesting another scenario,
// force safe occupancy context to AWAY while system remains in MODE_NORMAL.
IF VI_System_Mode = E_System_Operating_Mode.MODE_NORMAL THEN
    IF VI_Security_Armed AND
       (VIO_Scenario_Req_Operator = E_SCENARIO_TYPE.SCENARIO_NONE) AND
       (VIO_Scenario_Req_Gateway = E_SCENARIO_TYPE.SCENARIO_NONE) AND
       (VIO_Scenario_Req_Rule = E_SCENARIO_TYPE.SCENARIO_NONE) AND
       (VIO_Scenario_Intent <> E_SCENARIO_TYPE.SCENARIO_AWAY) THEN

        IF VIO_Scenario_Intent <> E_SCENARIO_TYPE.SCENARIO_AWAY THEN
            VIO_Scenario_Intent := E_SCENARIO_TYPE.SCENARIO_AWAY;
            VIO_Scenario_Source := SRC_POLICY;

            fbLogEvent(
                VI_Event_Type := 5,
                VI_Timestamp := VI_System_Time_MS,
                VI_Param1 := TO_UDINT(VIO_Scenario_Source),
                VI_Param2 := TO_UDINT(E_SCENARIO_TYPE.SCENARIO_AWAY)
            );
        END_IF;
    END_IF;
END_IF;

// === DEGRADED-AWARE SCENARIO ADAPTATION ===
// Soft adaptation in degraded mode: keep explicit requests intact,
// but if no source is requesting a scenario, move behavior to a safer baseline.
IF VI_System_Mode = E_System_Operating_Mode.MODE_DEGRADED THEN
    IF (VIO_Scenario_Req_Operator = E_SCENARIO_TYPE.SCENARIO_NONE) AND
       (VIO_Scenario_Req_Gateway = E_SCENARIO_TYPE.SCENARIO_NONE) AND
       (VIO_Scenario_Req_Rule = E_SCENARIO_TYPE.SCENARIO_NONE) THEN

        IF VI_Security_Armed THEN
            IF VIO_Scenario_Intent <> E_SCENARIO_TYPE.SCENARIO_AWAY THEN
                VIO_Scenario_Intent := E_SCENARIO_TYPE.SCENARIO_AWAY;
                VIO_Scenario_Source := SRC_POLICY;

                fbLogEvent(
                    VI_Event_Type := 6,
                    VI_Timestamp := VI_System_Time_MS,
                    VI_Param1 := TO_UDINT(VIO_Scenario_Source),
                    VI_Param2 := TO_UDINT(E_SCENARIO_TYPE.SCENARIO_AWAY)
                );
            END_IF;

        ELSIF VIO_Scenario_Intent = E_SCENARIO_TYPE.SCENARIO_PRESENCE THEN
            IF VIO_Scenario_Intent <> E_SCENARIO_TYPE.SCENARIO_SLEEP THEN
                VIO_Scenario_Intent := E_SCENARIO_TYPE.SCENARIO_SLEEP;
                VIO_Scenario_Source := SRC_POLICY;

                fbLogEvent(
                    VI_Event_Type := 7,
                    VI_Timestamp := VI_System_Time_MS,
                    VI_Param1 := TO_UDINT(VIO_Scenario_Source),
                    VI_Param2 := TO_UDINT(E_SCENARIO_TYPE.SCENARIO_SLEEP)
                );
            END_IF;
        END_IF;
    END_IF;
END_IF;

fbScenarioManager(
    VI_System_Time_MS := VI_System_Time_MS,
    VI_Activate_Request := VIO_Scenario_Intent,
    VI_IsActivePLC := VI_IsActivePLC,
    VI_System_Mode := VI_System_Mode,
    VO_Current_Scenario => GVL_STATUS.G_Current_Scenario
);

// >>> BULK_SYNC_ANCHOR: FB_System_Scenario_Arbitration <<<
          
END_FUNCTION_BLOCK

FUNCTION_BLOCK FB_Heating_Manifold_Control
  VAR_INPUT
    VI_System_Time_MS : UDINT;
    VI_IsActivePLC : BOOL;
    VI_DHW_Heating_Demand : BOOL;
    VI_Freeze_Mode_Active : BOOL;
    VI_Target_Supply_Temp : REAL;
    VI_Any_Zone_Active : ARRAY[1..GVL_CONSTANTS.C_MAX_MANIFOLDS] OF BOOL;
  END_VAR
  VAR_OUTPUT
    VO_Manifold_Pumps : ARRAY[1..GVL_CONSTANTS.C_MAX_MANIFOLDS] OF BOOL;
    VO_Manifold_Valves : ARRAY[1..GVL_CONSTANTS.C_MAX_MANIFOLDS] OF REAL;
    VO_Status : ARRAY[1..GVL_CONSTANTS.C_MAX_MANIFOLDS] OF ST_Manifold_Status;
  END_VAR
  VAR_IN_OUT
    VI_Manifold_Pressures : ARRAY[1..GVL_CONSTANTS.C_MAX_MANIFOLDS] OF REAL;
    VI_Manifold_Currents : ARRAY[1..GVL_CONSTANTS.C_MAX_MANIFOLDS] OF REAL;
    VI_Manifold_Temps_Supply : ARRAY[1..GVL_CONSTANTS.C_MAX_MANIFOLDS] OF REAL;
    VI_Manifold_Temps_Return : ARRAY[1..GVL_CONSTANTS.C_MAX_MANIFOLDS] OF REAL;
  END_VAR
  VAR
    L_i : INT;
    L_Delta_T : REAL;
    L_PID_Valves : ARRAY[1..GVL_CONSTANTS.C_MAX_MANIFOLDS] OF FB_PID_Controller;
    L_PID_Timer : ARRAY[1..GVL_CONSTANTS.C_MAX_MANIFOLDS] OF FB_System_Timer;
    L_Pump_Run_Timer : ARRAY[1..GVL_CONSTANTS.C_MAX_MANIFOLDS] OF FB_System_Timer;
    L_Pump_Pause_Timer : ARRAY[1..GVL_CONSTANTS.C_MAX_MANIFOLDS] OF FB_System_Timer;
    L_Pump_In_Pause : ARRAY[1..GVL_CONSTANTS.C_MAX_MANIFOLDS] OF BOOL;
    L_Pump_Diag : ARRAY[1..GVL_CONSTANTS.C_MAX_MANIFOLDS] OF FB_Device_Predictive_Diag;
  END_VAR

            // ==============================================================================
// Heating manifold control helper
// Internal refactoring helper for FB_Heating_System_Manager.
// Valve test override remains in FB_Heating_System_Manager for now.
// ==============================================================================



FOR L_i := 1 TO GVL_CONSTANTS.C_MAX_MANIFOLDS DO
    L_PID_Timer[L_i](IN := TRUE, PT := T#1s, VI_System_Time_MS := VI_System_Time_MS);
    IF L_PID_Timer[L_i].Q THEN
        L_PID_Timer[L_i](IN := FALSE, PT := T#1s, VI_System_Time_MS := VI_System_Time_MS);
        L_PID_Timer[L_i](IN := TRUE, PT := T#1s, VI_System_Time_MS := VI_System_Time_MS);

        L_PID_Valves[L_i](
            VI_SetPoint := VI_Target_Supply_Temp,
            VI_ProcessValue := VI_Manifold_Temps_Supply[L_i],
            VI_Kp := 2.0,
            VI_Tn := 120.0,
            VI_Tv := 0.0,
            VI_Y_Min := 0.0,
            VI_Y_Max := 100.0,
            VI_Cycle_Time_S := 1.0,
            VO_Output => VO_Manifold_Valves[L_i]
        );
    END_IF;

    L_Pump_Run_Timer[L_i](
        IN := VO_Manifold_Pumps[L_i] AND NOT L_Pump_In_Pause[L_i],
        PT := T#72h,
        VI_System_Time_MS := VI_System_Time_MS
    );
    IF L_Pump_Run_Timer[L_i].Q THEN
        L_Pump_In_Pause[L_i] := TRUE;
    END_IF;

    L_Pump_Pause_Timer[L_i](
        IN := L_Pump_In_Pause[L_i],
        PT := T#1h,
        VI_System_Time_MS := VI_System_Time_MS
    );
    IF L_Pump_Pause_Timer[L_i].Q THEN
        L_Pump_In_Pause[L_i] := FALSE;
    END_IF;

    IF VI_DHW_Heating_Demand THEN
        VO_Manifold_Pumps[L_i] := FALSE;
        VO_Manifold_Valves[L_i] := 0.0;
    ELSE
        VO_Manifold_Pumps[L_i] := VI_IsActivePLC AND VI_Any_Zone_Active[L_i] AND NOT L_Pump_In_Pause[L_i];
    END_IF;

    IF VI_Freeze_Mode_Active THEN
        VO_Manifold_Pumps[L_i] := TRUE;
        IF VO_Manifold_Valves[L_i] < 35.0 THEN
            VO_Manifold_Valves[L_i] := 35.0;
        END_IF;
    END_IF;

    VO_Status[L_i].Pump_On := VO_Manifold_Pumps[L_i];
    VO_Status[L_i].Pump_Current := VI_Manifold_Currents[L_i];
    VO_Status[L_i].Pressure := VI_Manifold_Pressures[L_i];
    VO_Status[L_i].Temp_Supply := VI_Manifold_Temps_Supply[L_i];
    VO_Status[L_i].Temp_Return := VI_Manifold_Temps_Return[L_i];
    VO_Status[L_i].Valve_Pos := VO_Manifold_Valves[L_i];

    L_Pump_Diag[L_i](
        VI_Current_Value := VI_Manifold_Currents[L_i],
        VI_Nominal_Value := 0.55,
        VI_Is_Running := VO_Manifold_Pumps[L_i],
        VI_Reset_Stats := FALSE,
        VI_System_Time_MS := VI_System_Time_MS,
        VIO_Health_Data := VO_Status[L_i].Health
    );

    IF VO_Manifold_Pumps[L_i] THEN
        L_Delta_T := VI_Manifold_Temps_Supply[L_i] - VI_Manifold_Temps_Return[L_i];

        VO_Status[L_i].Error := FALSE;
        VO_Status[L_i].Error_ID := 0;

        IF VI_Manifold_Currents[L_i] <= 0.01 THEN
            VO_Status[L_i].Error := TRUE;
            VO_Status[L_i].Error_ID := TO_WORD(GVL_CONFIG.ERR_PUMP_NO_CURRENT);
        ELSIF VI_Manifold_Currents[L_i] < 0.3 THEN
            VO_Status[L_i].Error := TRUE;
            VO_Status[L_i].Error_ID := TO_WORD(GVL_CONFIG.ERR_PUMP_UNDERCURRENT);
        ELSIF VI_Manifold_Currents[L_i] > 1.5 THEN
            VO_Status[L_i].Error := TRUE;
            VO_Status[L_i].Error_ID := TO_WORD(GVL_CONFIG.ERR_PUMP_OVERCURRENT);
        END_IF;

        IF (NOT VO_Status[L_i].Error) AND ((VI_Manifold_Pressures[L_i] < 1.5) OR (VI_Manifold_Pressures[L_i] > 2.5)) THEN
            VO_Status[L_i].Error := TRUE;
            VO_Status[L_i].Error_ID := TO_WORD(GVL_CONFIG.ERR_PRESSURE_OUT_OF_RANGE);
        END_IF;

        IF NOT VO_Status[L_i].Error THEN
            IF L_Delta_T < 5.0 THEN
                VO_Status[L_i].Error := TRUE;
                VO_Status[L_i].Error_ID := TO_WORD(GVL_CONFIG.ERR_DELTA_T_LOW);
            ELSIF L_Delta_T > 10.0 THEN
                VO_Status[L_i].Error := TRUE;
                VO_Status[L_i].Error_ID := TO_WORD(GVL_CONFIG.ERR_DELTA_T_HIGH);
            END_IF;
        END_IF;
    END_IF;
END_FOR;

// >>> BULK_SYNC_ANCHOR: FB_Heating_Manifold_Control <<<
          
END_FUNCTION_BLOCK

